(*************************************************************
This function was generated by the 'check array access'
option of the controllers 'properties' dialog box.
If you delete this comment, the 'check array access' option
of the controllers 'properties' dialog box will be removed.
**************************************************************)
    (**************************************************************************************************)
    (* The implementation has to be adjusted to your application/machine.                             *)
    (* This is an exemplary implementation of the function.                                           *)
    (* Per default, an access violation is generated to avoid machine damage                          *)
    (* Check the Call Stack (menu Debug/Callstack) and modify the faulty logic!                       *)
    (**************************************************************************************************)

IF  index < lower THEN 
	errstr:= 'CheckBounds: Lower arrayindex ';
	errstr:=CONCAT(STR1:=errstr  , STR2:= DINT_TO_STRING(lower));
	errstr:=CONCAT(STR1:=errstr  , STR2:= ' underrunned by ');
	errstr:=CONCAT(STR1:=errstr  , STR2:= DINT_TO_STRING(index));
//  This pragma may be removed: 
	{info 'CheckBounds: Please implement your own error reaction below'}
//  EXAMPLE 1 (default): 
//  Set a F0-Error into the diagnostic- and error memory
//  Triggering an access violation --> Application will be stopped and leads to a F5-Error

  ML_SetDiagEntry(
	Severity:= E_LOG_SEVERITY.ERROR, 
	Class:= E_LOG_CLASS.CLASS_0, 
	Facility:= E_LOG_FACILITY.USER, 
	Code:= 0, 
	Text:= ADR(errstr));

	bByte:=ptNull^;(*triggering an access violation *)

// EXAMPLE 2:
// Limit the faulty index to the lower index 
//     -> no memory will be overwritten
//     -> Keep PLC-task and motion running
// Set a E0-Warning into the diagnostic- and error memory
// NOTE: There is still an implementation error in your application code!

//  ML_SetDiagEntry(
//	Severity:= E_LOG_SEVERITY.WARNING, 
//	Class:= E_LOG_CLASS.CLASS_0, 
//	Facility:= E_LOG_FACILITY.USER, 
//	Code:= 0, 
//	Text:= ADR(errstr));
// 
//	CheckBounds := lower; //access to the lower index only 
//  return;
	
ELSIF  index > upper THEN
	errstr:= 'CheckBounds: Higher arrayindex ';
	errstr:=CONCAT(STR1:=errstr  , STR2:= DINT_TO_STRING(upper));
	errstr:=CONCAT(STR1:=errstr  , STR2:= ' overrunned by ');
	errstr:=CONCAT(STR1:=errstr  , STR2:= DINT_TO_STRING(index));

//  this pragma may be removed: 
	{info 'CheckBounds: Please implement your own error reaction below'}
//  example 1 (default): 
//  set a F0-Error into the diagnostic- and error memory
//  triggering an access violation --> Application will be stopped and leads to a F5-Error

  ML_SetDiagEntry(
	Severity:= E_LOG_SEVERITY.ERROR, 
	Class:= E_LOG_CLASS.CLASS_0, 
	Facility:= E_LOG_FACILITY.USER, 
	Code:= 0, 
	Text:= ADR(errstr));

	bByte:=ptNull^;(*triggering an access violation *)

//example 2:
// Limit the faulty index to the upper index 
//     -> no memory will be overwritten
//     -> Keep PLC-task and motion running
// Set a E0-Warning into the diagnostic- and error memory
// NOTE: There is still an implementation error in your application code!

//  ML_SetDiagEntry(
//	Severity:= E_LOG_SEVERITY.WARNING, 
//	Class:= E_LOG_CLASS.CLASS_0, 
//	Facility:= E_LOG_FACILITY.USER, 
//	Code:= 0, 
//	Text:= ADR(errstr));
// 
//	CheckBounds := upper; //access to the upper index only 
//  return;

ELSE // access to array is ok  
	CheckBounds := index;
END_IF

END_FUNCTION

// IndraMotionMlc1/Application/Discrete_FIlter
FUNCTION_BLOCK Discrete_FIlter
VAR_INPUT
	ssMethodType: SINT;
	In: LREAL;
END_VAR
VAR_OUTPUT
	Out: LREAL;
END_VAR
VAR
	DiscreteFilter_states: LREAL;
END_VAR



CASE ssMethodType OF
    0: 
        (* InitializeConditions for DiscreteFilter: '<S1>/Discrete Filter' *)
        DiscreteFilter_states := 0.0;
    1: 
        (* DiscreteFilter: '<S1>/Discrete Filter' *)
        Out := In - (0.5 * DiscreteFilter_states);
        (* Update for DiscreteFilter: '<S1>/Discrete Filter' *)
        DiscreteFilter_states := Out;
END_CASE;

END_FUNCTION_BLOCK

// IndraMotionMlc1/Application/VCC_Anti_DB
PROGRAM VCC_Anti_DB
VAR_INPUT
	u_ref: LREAL;
END_VAR
VAR_OUTPUT
	u_cmd:  LREAL := 6;
END_VAR
VAR
	cyl_extract: LREAL;
	cyl_retract: LREAL;
END_VAR

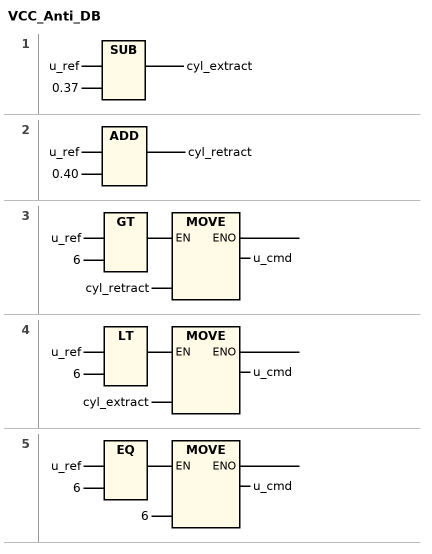
// NETWORK 1
cyl_extract := u_ref - 0.37;

// NETWORK 2
cyl_retract := u_ref + 0.40;

// NETWORK 3
IF u_ref > 6 THEN u_cmd := cyl_retract; END_IF

// NETWORK 4
IF u_ref < 6 THEN u_cmd := cyl_extract; END_IF

// NETWORK 5
IF u_ref = 6 THEN u_cmd := 6; END_IF

END_PROGRAM

// IndraMotionMlc1/Application/S_shape_Profile_old
FUNCTION_BLOCK S_shape_Profile_old
VAR_INPUT
	Enable: BOOL;
	x0: LREAL;
	v0: LREAL;
	Position_SP: LREAL;
	Velocity_SP: LREAL;
	t0: LREAL;
	t_Hold_Position: LREAL;
	CyclicTime: LREAL;
END_VAR
VAR_OUTPUT
	Position_Ref: LREAL;
	Velocity_Ref: LREAL;
	Motion_Cycle_Time: LREAL;
	Error: LREAL;
END_VAR
VAR
	Error_0: DINT;
	jm: LREAL;
	s_acc: LREAL;
	t1: LREAL;
	t2: LREAL;
	t3: LREAL;
	t4: LREAL;
	t5: LREAL;
	t6: LREAL;
	t7: LREAL;
	t8: LREAL;
	t9: LREAL;
	t10: LREAL;
	sh: LREAL;
	vh: LREAL;
	s3: LREAL;
	s4: LREAL;
	v4: LREAL;
	s7: LREAL;
	rtb_Saturation: LREAL;
	rtb_Saturation_tmp: LREAL;
END_VAR


(* Saturate: '<S1>/Saturation' *)

IF Position_SP >= 500.0 THEN 
    rtb_Saturation := 500.0;
ELSIF Position_SP > 0.0 THEN 
    rtb_Saturation := Position_SP;
ELSE 
    rtb_Saturation := 0.0;
END_IF;

(* End of Saturate: '<S1>/Saturation' *)


(* Saturate: '<S1>/Saturation1' *)

IF Velocity_SP >= 150.0 THEN 
    Position_Ref := 150.0;
ELSIF Velocity_SP > -150.0 THEN 
    Position_Ref := Velocity_SP;
ELSE 
    Position_Ref := -150.0;
END_IF;

(* End of Saturate: '<S1>/Saturation1' *)


(* MATLAB Function: '<S1>/SP_Generator' *)
(* MATLAB Function 'S_shape_Profile/SP_Generator': '<S2>:1' *)
(* '<S2>:1:4' PositionSP = Desired_Position - s0; *)
(* '<S2>:1:6' a0 = 0; *)
(* '<S2>:1:7' j0 = 0; *)
(* '<S2>:1:8' AccelerationSP = VelocitySP; *)
(* '<S2>:1:10' vel=VelocitySP; *)
(* '<S2>:1:11' as=AccelerationSP; *)
(* Input velocity  *)
(* '<S2>:1:13' vs=vel; *)
(* [rad/s] *)
(* Delta velocity  *)
(* '<S2>:1:15' dv=(vs-v0); *)
(* [rad/s]      *)
(* Max Jerk Considerations *)
(* '<S2>:1:17' jm=as^2/dv; *)
sh := Position_Ref * Position_Ref;
vh := Position_Ref - v0;
jm := sh / vh;
(* [rad/s^3]  *)
(* Constant Velocity periodes *)
(* '<S2>:1:19' s_acc=(vs^2-v0^2)/as; *)
s_acc := (sh - (v0 * v0)) / Position_Ref;
(* '<S2>:1:20' CstVelTime=(PositionSP-2*s_acc)/vs; *)
rtb_Saturation := ((rtb_Saturation - x0) - (2.0 * s_acc)) / Position_Ref;
(* '<S2>:1:21' if CstVelTime < 0 *)

IF rtb_Saturation < 0.0 THEN 
    (* '<S2>:1:22' Error = 1; *)
    Error_0 := 1;
ELSE 
    (* '<S2>:1:23' else *)
    (* '<S2>:1:24' Error = 0; *)
    Error_0 := 0;
END_IF;

(* Time periodes, *)
(* '<S2>:1:28' t1=t0+(as/jm); *)
s3 := Position_Ref / jm;
t1 := s3 + t0;
(* '<S2>:1:29' t2=t1+(as/jm); *)
t2 := s3 + t1;
(* '<S2>:1:30' t3=t2+CstVelTime; *)
t3 := t2 + rtb_Saturation;
(* '<S2>:1:31' t4=t3+(as/jm); *)
t4 := s3 + t3;
(* '<S2>:1:32' t5=t4+(as/jm); *)
t5 := s3 + t4;
(* '<S2>:1:33' t6=t5+HoldPositionTime; *)
t6 := t5 + t_Hold_Position;
(* '<S2>:1:34' t7=t6+(as/jm); *)
t7 := s3 + t6;
(* '<S2>:1:35' t8=t7+(as/jm); *)
t8 := s3 + t7;
(* '<S2>:1:36' t9=t8+CstVelTime; *)
t9 := t8 + rtb_Saturation;
(* '<S2>:1:37' t10=t9+(as/jm); *)
t10 := s3 + t9;
(* '<S2>:1:38' t11=t10+(as/jm); *)
Motion_Cycle_Time := s3 + t10;
(* Position and Velocity Constants *)
(* '<S2>:1:40' sh=(v0+(as^2)/(6*jm))*(as/jm); *)
sh := ((sh / (6.0 * jm)) + v0) * s3;
(* '<S2>:1:41' vh=(vs-v0)/2; *)
vh := vh / 2.0;
(* '<S2>:1:42' s3=s_acc+vs*(t3-t2); *)
s3 := ((t3 - t2) * Position_Ref) + s_acc;
(* '<S2>:1:43' s4=s3+vs*(t4-t3)-jm*((t4-t3)^3)/6; *)
rtb_Saturation := t4 - t3;
s4 := ((rtb_Saturation * Position_Ref) + s3) - ((EXPT(rtb_Saturation, 3.0) * jm) / 6.0);
(* '<S2>:1:44' v4=vs-jm*((t4-t3)^2)/2; *)
v4 := Position_Ref - (((rtb_Saturation * rtb_Saturation) * jm) / 2.0);
(* '<S2>:1:45' s5=s0+jm*((t5-t4)^3)/6-as*((t5-t4)^2)/2+v4*(t5-t4)+s4; *)
rtb_Saturation_tmp := t5 - t4;
rtb_Saturation := (((((EXPT(rtb_Saturation_tmp, 3.0) * jm) / 6.0) + x0) - (((rtb_Saturation_tmp * rtb_Saturation_tmp) * Position_Ref) / 2.0)) + (rtb_Saturation_tmp * v4)) + s4;
(* s6=s5+(s0+v0*(t7-t6)+jm*((t7-t6)^3)/6); *)
(* '<S2>:1:47' s7= s5-(s_acc+vs*(t9-t8)); *)
s7 := rtb_Saturation - (((t9 - t8) * Position_Ref) + s_acc);
(* '<S2>:1:48' s8= s7-(vs*(t10-t9)-jm*((t10-t9)^3)/6); *)
(* s9= s8-(jm*((t11-t10)^3)/6-as*((t11-t10)^2)/2+v4*(t11-t10)); *)
(* Phase0 *)
(* '<S2>:1:51' if  Error == 1 *)

IF Error_0 = 1 THEN 
    (* '<S2>:1:52' s = s0; *)
    rtb_Saturation := x0;
    (* '<S2>:1:53' v = v0; *)
    Position_Ref := v0;
    (* '<S2>:1:54' a = a0; *)
    (* '<S2>:1:55' j=j0; *)
ELSIF (CyclicTime >= 0.0) AND (CyclicTime <= t0) THEN 
    (* '<S2>:1:56' elseif  (t >= 0) &amp;&amp; (t <= t0) *)
    (* '<S2>:1:57' s = s0; *)
    rtb_Saturation := x0;
    (* '<S2>:1:58' v = v0; *)
    Position_Ref := v0;
    (* '<S2>:1:59' a = a0; *)
    (* '<S2>:1:60' j=j0; *)
    (* Phase1 - concave Acc *)
ELSIF (CyclicTime >= t0) AND (CyclicTime <= t1) THEN 
    (* '<S2>:1:62' elseif  (t >= t0) &amp;&amp; (t <= (t1)) *)
    (* '<S2>:1:63' s = s0+v0*(t-t0)+jm*((t-t0)^3)/6; *)
    rtb_Saturation_tmp := CyclicTime - t0;
    rtb_Saturation := ((rtb_Saturation_tmp * v0) + x0) + ((EXPT(rtb_Saturation_tmp, 3.0) * jm) / 6.0);
    (* '<S2>:1:64' v = v0+jm*((t-t0)^2)/2; *)
    Position_Ref := (((rtb_Saturation_tmp * rtb_Saturation_tmp) * jm) / 2.0) + v0;
    (* '<S2>:1:65' a = jm*(t-t0); *)
    (* '<S2>:1:66' j=jm; *)
    (* Phase2 - convex Acc *)
ELSIF (CyclicTime >= t1) AND (CyclicTime <= t2) THEN 
    (* '<S2>:1:68' elseif (t >= (t1)) &amp;&amp; (t <= (t2)) *)
    (* '<S2>:1:69' s = s0+sh+vh*(t-t1)+as*((t-t1)^2)/2-jm*((t-t1)^3)/6; *)
    rtb_Saturation_tmp := CyclicTime - t1;
    rtb_Saturation := (((rtb_Saturation_tmp * vh) + (x0 + sh)) + (((rtb_Saturation_tmp * rtb_Saturation_tmp) * Position_Ref) / 2.0)) - ((EXPT(rtb_Saturation_tmp, 3.0) * jm) / 6.0);
    (* '<S2>:1:70' v = vh+as*(t-t1)-jm*((t-t1)^2)/2; *)
    Position_Ref := ((rtb_Saturation_tmp * Position_Ref) + vh) - (((rtb_Saturation_tmp * rtb_Saturation_tmp) * jm) / 2.0);
    (* '<S2>:1:71' a = as-jm*(t-t1); *)
    (* '<S2>:1:72' j = -jm; *)
    (* Phase3 - constant velocity *)
ELSIF (CyclicTime >= t2) AND (CyclicTime <= t3) THEN 
    (* '<S2>:1:74' elseif (t >= t2) &amp;&amp; (t <= t3) *)
    (* '<S2>:1:75' s = s0+s_acc+vs*(t-t2); *)
    rtb_Saturation := ((CyclicTime - t2) * Position_Ref) + (x0 + s_acc);
    (* '<S2>:1:76' v = vs; *)
    (* '<S2>:1:77' a = 0; *)
    (* '<S2>:1:78' j = 0; *)
    (* Phase4 - convex Dec *)
ELSIF (CyclicTime >= t3) AND (CyclicTime <= t4) THEN 
    (* '<S2>:1:80' elseif (t >= t3) &amp;&amp; (t <= t4) *)
    (* '<S2>:1:81' s = s0+s3+vs*(t-t3)-jm*((t-t3)^3)/6; *)
    rtb_Saturation_tmp := CyclicTime - t3;
    rtb_Saturation := ((rtb_Saturation_tmp * Position_Ref) + (x0 + s3)) - ((EXPT(rtb_Saturation_tmp, 3.0) * jm) / 6.0);
    (* '<S2>:1:82' v = vs-jm*((t-t3)^2)/2; *)
    Position_Ref := Position_Ref - (((rtb_Saturation_tmp * rtb_Saturation_tmp) * jm) / 2.0);
    (* '<S2>:1:83' a = -jm*(t-t3); *)
    (* '<S2>:1:84' j = -jm; *)
    (* Phase5 - concav Dec *)
ELSIF (CyclicTime >= t4) AND (CyclicTime <= t5) THEN 
    (* '<S2>:1:86' elseif (t >= t4) &amp;&amp; (t <= t5) *)
    (* '<S2>:1:87' s = s0+jm*((t-t4)^3)/6-as*((t-t4)^2)/2+v4*(t-t4)+s4; *)
    rtb_Saturation_tmp := CyclicTime - t4;
    rtb_Saturation := (((((EXPT(rtb_Saturation_tmp, 3.0) * jm) / 6.0) + x0) - (((rtb_Saturation_tmp * rtb_Saturation_tmp) * Position_Ref) / 2.0)) + (rtb_Saturation_tmp * v4)) + s4;
    (* '<S2>:1:88' v = jm*((t-t4)^2)/2-as*(t-t4)+v4; *)
    Position_Ref := ((((rtb_Saturation_tmp * rtb_Saturation_tmp) * jm) / 2.0) - (rtb_Saturation_tmp * Position_Ref)) + v4;
    (* '<S2>:1:89' a = jm*(t-t4)-as; *)
    (* '<S2>:1:90' j=jm; *)
    (* Phase6 - holding position *)
ELSIF (CyclicTime >= t5) AND (CyclicTime <= t6) THEN 
    (* '<S2>:1:92' elseif (t >= t5) &amp;&amp; (t <= t6) *)
    (* '<S2>:1:93' s = s5; *)
    (* '<S2>:1:94' v = 0; *)
    Position_Ref := 0.0;
    (* '<S2>:1:95' a = 0; *)
    (* '<S2>:1:96' j = 0; *)
    (* Phase7 - concave Dec *)
ELSIF (CyclicTime >= t6) AND (CyclicTime <= t7) THEN 
    (* '<S2>:1:98' elseif (t >= t6) &amp;&amp; (t <= t7) *)
    (* '<S2>:1:99' s = s5-(v0*(t-t6)+jm*((t-t6)^3)/6); *)
    rtb_Saturation_tmp := CyclicTime - t6;
    rtb_Saturation := rtb_Saturation - (((EXPT(rtb_Saturation_tmp, 3.0) * jm) / 6.0) + (rtb_Saturation_tmp * v0));
    (* '<S2>:1:100' v = -(v0+jm*((t-t6)^2)/2); *)
    Position_Ref :=  -((((rtb_Saturation_tmp * rtb_Saturation_tmp) * jm) / 2.0) + v0);
    (* '<S2>:1:101' a = -jm*(t-t6); *)
    (* '<S2>:1:102' j=-jm; *)
    (* Phase8 - convex Dec *)
ELSIF (CyclicTime >= t7) AND (CyclicTime <= t8) THEN 
    (* '<S2>:1:104' elseif (t >= t7) &amp;&amp; (t <= t8) *)
    (* '<S2>:1:105' s = s5-(sh+vh*(t-t7)+as*((t-t7)^2)/2-jm*((t-t7)^3)/6); *)
    s3 := CyclicTime - t7;
    rtb_Saturation := rtb_Saturation - ((((s3 * vh) + sh) + (((s3 * s3) * Position_Ref) / 2.0)) - ((EXPT(s3, 3.0) * jm) / 6.0));
    (* '<S2>:1:106' v = -(vh+as*(t-t7)-jm*((t-t7)^2)/2); *)
    Position_Ref :=  -(((s3 * Position_Ref) + vh) - (((s3 * s3) * jm) / 2.0));
    (* '<S2>:1:107' a = -(as-jm*(t-t7)); *)
    (* '<S2>:1:108' j = jm; *)
    (* Phase9 - constant velocity *)
ELSIF (CyclicTime >= t8) AND (CyclicTime <= t9) THEN 
    (* '<S2>:1:110' elseif (t >= t8) &amp;&amp; (t <= t9) *)
    (* '<S2>:1:111' s = s5-(s_acc+vs*(t-t8)); *)
    rtb_Saturation := rtb_Saturation - (((CyclicTime - t8) * Position_Ref) + s_acc);
    (* '<S2>:1:112' v = -vs; *)
    Position_Ref :=  -Position_Ref;
    (* '<S2>:1:113' a = 0; *)
    (* '<S2>:1:114' j = 0; *)
    (* Phase10 - concav Acc *)
ELSIF (CyclicTime >= t9) AND (CyclicTime <= t10) THEN 
    (* '<S2>:1:116' elseif (t >= t9) &amp;&amp; (t <= t10) *)
    (* '<S2>:1:117' s = s7-(vs*(t-t9)-jm*((t-t9)^3)/6); *)
    rtb_Saturation_tmp := CyclicTime - t9;
    rtb_Saturation := s7 - ((rtb_Saturation_tmp * Position_Ref) - ((EXPT(rtb_Saturation_tmp, 3.0) * jm) / 6.0));
    (* '<S2>:1:118' v = -(vs-jm*((t-t9)^2)/2); *)
    Position_Ref :=  -(Position_Ref - (((rtb_Saturation_tmp * rtb_Saturation_tmp) * jm) / 2.0));
    (* '<S2>:1:119' a = jm*(t-t9); *)
    (* '<S2>:1:120' j = jm; *)
    (* Phase11 - convex Acc *)
ELSIF (CyclicTime >= t10) AND (CyclicTime <= Motion_Cycle_Time) THEN 
    (* '<S2>:1:122' elseif (t >= t10) &amp;&amp; (t <= t11) *)
    (* '<S2>:1:123' s = s8-(jm*((t-t10)^3)/6-as*((t-t10)^2)/2+v4*(t-t10)); *)
    rtb_Saturation_tmp := CyclicTime - t10;
    rtb_Saturation := t10 - t9;
    rtb_Saturation := (s7 - ((rtb_Saturation * Position_Ref) - ((EXPT(rtb_Saturation, 3.0) * jm) / 6.0))) - ((((EXPT(rtb_Saturation_tmp, 3.0) * jm) / 6.0) - (((rtb_Saturation_tmp * rtb_Saturation_tmp) * Position_Ref) / 2.0)) + (rtb_Saturation_tmp * v4));
    (* '<S2>:1:124' v = -(jm*((t-t10)^2)/2-as*(t-t10)+v4); *)
    Position_Ref :=  -(((((rtb_Saturation_tmp * rtb_Saturation_tmp) * jm) / 2.0) - (rtb_Saturation_tmp * Position_Ref)) + v4);
    (* '<S2>:1:125' a = -(jm*(t-t10)-as); *)
    (* '<S2>:1:126' j=-jm; *)
    (* Phase12 - hold position *)
ELSE 
    (* '<S2>:1:128' else *)
    (* '<S2>:1:129' s = s0; *)
    rtb_Saturation := x0;
    (* '<S2>:1:130' v = v0; *)
    Position_Ref := v0;
    (* '<S2>:1:131' a = a0; *)
    (* '<S2>:1:132' j = j0; *)
END_IF;

(* '<S2>:1:135' if t == 0 *)

IF CyclicTime = 0.0 THEN 
    (* '<S2>:1:136' PositionRef=s0; *)
    rtb_Saturation := x0;
    (* [mm] *)
END_IF;

(* Switch: '<S1>/Switch' *)
(* '<S2>:1:141' InPositionTime=t11; *)
(* [s] *)
(* '<S2>:1:142' VelocityRef=v; *)
(* [mm/s] *)
(* '<S2>:1:143' AccelerationRef=a; *)
(* [mm/s^2] *)
(* '<S2>:1:144' JerkRef=j; *)
(* %[mm/s^3] *)

IF  NOT Enable THEN 
    Position_Ref := v0;
END_IF;

(* End of Switch: '<S1>/Switch' *)


(* Saturate: '<S1>/Saturation2' *)

IF Position_Ref >= 150.0 THEN 
    (* Outport: '<Root>/Velocity_Ref' *)
    Velocity_Ref := 150.0;
ELSIF Position_Ref > -150.0 THEN 
    (* Outport: '<Root>/Velocity_Ref' *)
    Velocity_Ref := Position_Ref;
ELSE 
    (* Outport: '<Root>/Velocity_Ref' *)
    Velocity_Ref := -150.0;
END_IF;

(* End of Saturate: '<S1>/Saturation2' *)


(* Switch: '<S1>/Switch1' *)

IF Enable THEN 
    Position_Ref := rtb_Saturation;
ELSE 
    Position_Ref := x0;
END_IF;

(* End of Switch: '<S1>/Switch1' *)


(* Saturate: '<S1>/Saturation3' *)

IF Position_Ref >= 500.0 THEN 
    (* Outport: '<Root>/Position_Ref' *)
    Position_Ref := 500.0;
ELSIF  NOT (Position_Ref > 0.0) THEN 
    (* Outport: '<Root>/Position_Ref' *)
    Position_Ref := 0.0;
END_IF;

(* End of Saturate: '<S1>/Saturation3' *)


(* Outport: '<Root>/Error' incorporates:
 *  MATLAB Function: '<S1>/SP_Generator' *)
Error := DINT_TO_LREAL(Error_0);

END_FUNCTION_BLOCK

// IndraMotionMlc1/Application/VCC_Controller_FF_PI_AD_v04
FUNCTION_BLOCK VCC_Controller_FF_PI_AD_v04
VAR_INPUT
	ssMethodType: SINT;
	Tuning_Mode_On: BOOL;
	FB_Cntr_On: BOOL;
	I_Cntr_On: BOOL;
	I_Cntr_Reset_On: BOOL;
	Active_Damper_On: BOOL;
	k_AD_Num: LREAL;
	Pos_Error_Limit: LREAL;
	DB_Up: LREAL;
	DB_Down: LREAL;
	Qmax_Up: LREAL;
	Qmax_Down: LREAL;
	k_P: LREAL;
	k_I: LREAL;
	Pos_Ref: LREAL;
	Vel_Ref: LREAL;
	Pos_FB: LREAL;
	p_A: LREAL;
	p_B: LREAL;
END_VAR
VAR_OUTPUT
	Pos_Error: LREAL;
	u_FF: LREAL;
	u_P: LREAL;
	u_I: LREAL;
	u_AD: LREAL;
	I_reset: LREAL;
	u_DCV: LREAL;
END_VAR
VAR
	rtb_Q_refm3s: LREAL;
	rtb_Saturation1: LREAL;
	rtb_I_Reset: DINT;
	rtb_LoadPressure: LREAL;
	c_DiscreteTimeIntegrator_DS: LREAL;
	VectorConcatenate: ARRAY[0..1] OF LREAL;
	TransferFcn11_states: LREAL;
END_VAR



CASE ssMethodType OF
    0: 
        (* InitializeConditions for DiscreteIntegrator: '<S1>/Discrete-Time Integrator' *)
        c_DiscreteTimeIntegrator_DS := 0.0;
        (* InitializeConditions for DiscreteTransferFcn: '<S4>/Transfer Fcn1 1' *)
        TransferFcn11_states := 0.0;
    1: 
        (* Switch: '<S1>/Switch2' incorporates:
         *  Constant: '<S1>/Annnulus_Area'
         *  Constant: '<S1>/Bore_Area'
         *  Product: '<S1>/Product1'
         *  Product: '<S1>/Product3' *)

        IF Vel_Ref >= 0.0 THEN 
            u_FF := 3318.3 * Vel_Ref;
        ELSE 
            u_FF := Vel_Ref * 2356.2;
        END_IF;

        (* End of Switch: '<S1>/Switch2' *)
        

        (* Gain: '<S1>/Gain2' *)
        rtb_Q_refm3s := 1.0E-9 * u_FF;
        (* Switch: '<S1>/Switch5' *)

        IF Vel_Ref >= 0.0 THEN 
            u_FF := Qmax_Up;
        ELSE 
            u_FF := Qmax_Down;
        END_IF;

        (* End of Switch: '<S1>/Switch5' *)
        

        (* Product: '<S1>/Divide2' incorporates:
         *  Gain: '<S1>/Gain1' *)
        u_FF := (60000.0 * rtb_Q_refm3s) / u_FF;
        (* Sum: '<S1>/Sum1' *)
        Pos_Error := Pos_Ref - Pos_FB;
        (* Product: '<S1>/Product' *)
        u_P := k_P * Pos_Error;
        (* MATLAB Function: '<S1>/Controller_Reset' *)
        (* MATLAB Function 'VCC_Controller_FF_PI_AD_v04/Controller_Reset': '<S3>:1' *)
        (* '<S3>:1:3' I_Reset = 1; *)
        (* '<S3>:1:5' if (abs(Pos_Error) <= Pos_Error_Limit) &amp;&amp; (Vel_SP == 0) *)

        IF ABS(Pos_Error) <= Pos_Error_Limit THEN 

            IF Vel_Ref = 0.0 THEN 
                (* '<S3>:1:6' I_Reset = 1; *)
                rtb_I_Reset := 1;
            ELSE 
                (* '<S3>:1:7' else *)
                (* '<S3>:1:8' I_Reset = 0; *)
                rtb_I_Reset := 0;
            END_IF;

        ELSE 
            (* '<S3>:1:7' else *)
            (* '<S3>:1:8' I_Reset = 0; *)
            rtb_I_Reset := 0;
        END_IF;

        (* End of MATLAB Function: '<S1>/Controller_Reset' *)
        

        (* Switch: '<S1>/Switch3' incorporates:
         *  Constant: '<S1>/Constant2' *)

        IF I_Cntr_Reset_On THEN 
            I_reset := DINT_TO_LREAL(rtb_I_Reset);
        ELSE 
            I_reset := 0.0;
        END_IF;

        (* End of Switch: '<S1>/Switch3' *)
        

        (* DiscreteIntegrator: '<S1>/Discrete-Time Integrator' *)

        IF I_reset <> 0.0 THEN 
            c_DiscreteTimeIntegrator_DS := 0.0;
        END_IF;

        (* SignalConversion: '<S4>/ConcatBufferAtVector ConcatenateIn1' *)
        VectorConcatenate[0] := k_AD_Num;
        (* Gain: '<S4>/Gain1' *)
        VectorConcatenate[1] :=  -k_AD_Num;
        (* DiscreteTransferFcn: '<S4>/Transfer Fcn1 1' incorporates:
         *  Gain: '<S4>/Cylinder Area Ratio'
         *  Sum: '<S4>/Load Pressure' *)
        rtb_Q_refm3s := (p_A - (0.710059171597633 * p_B)) - (-0.997 * TransferFcn11_states);
        u_AD := (VectorConcatenate[0] * rtb_Q_refm3s) + (VectorConcatenate[1] * TransferFcn11_states);
        (* Switch: '<S1>/Switch' incorporates:
         *  Constant: '<S1>/Constant'
         *  DiscreteIntegrator: '<S1>/Discrete-Time Integrator' *)

        IF I_Cntr_On THEN 
            u_I := c_DiscreteTimeIntegrator_DS;
        ELSE 
            u_I := 0.0;
        END_IF;

        (* End of Switch: '<S1>/Switch' *)
        

        (* Switch: '<S1>/Switch1' incorporates:
         *  Constant: '<S1>/Constant1'
         *  Sum: '<S1>/Sum5' *)

        IF FB_Cntr_On THEN 
            rtb_LoadPressure := u_P + u_I;
        ELSE 
            rtb_LoadPressure := 0.0;
        END_IF;

        (* End of Switch: '<S1>/Switch1' *)
        

        (* Saturate: '<S1>/Saturation1' *)

        IF rtb_LoadPressure >= 1.0 THEN 
            rtb_Saturation1 := 1.0;
        ELSIF rtb_LoadPressure > -1.0 THEN 
            rtb_Saturation1 := rtb_LoadPressure;
        ELSE 
            rtb_Saturation1 := -1.0;
        END_IF;

        (* End of Saturate: '<S1>/Saturation1' *)
        

        (* Switch: '<S1>/Switch4' incorporates:
         *  Constant: '<S1>/Constant3' *)

        IF  NOT Active_Damper_On THEN 
            u_AD := 0.0;
        END_IF;

        (* End of Switch: '<S1>/Switch4' *)
        

        (* Gain: '<S1>/Gain' incorporates:
         *  Sum: '<S1>/Sum6' *)
        u_DCV :=  -((u_FF + rtb_Saturation1) - u_AD);
        (* Saturate: '<S1>/Saturation5' *)

        IF u_DCV >= 1.0 THEN 
            u_DCV := 1.0;
        ELSIF  NOT (u_DCV > -1.0) THEN 
            u_DCV := -1.0;
        END_IF;

        (* End of Saturate: '<S1>/Saturation5' *)
        

        (* MATLAB Function: '<S1>/Anti_Dead_Band' *)
        (* MATLAB Function 'VCC_Controller_FF_PI_AD_v04/Anti_Dead_Band': '<S2>:1' *)
        (* '<S2>:1:5' u_DCV = 0; *)
        (* '<S2>:1:7' if (I_Reset == 1) &amp;&amp; (Tuning_Mode == 0) *)

        IF (rtb_I_Reset = 1) AND ( NOT Tuning_Mode_On) THEN 
            (* Outport: '<Root>/u_DCV' *)
            (* '<S2>:1:8' u_DCV = 0; *)
            u_DCV := 0.0;
        ELSIF u_DCV < -0.001 THEN 
            (* Outport: '<Root>/u_DCV' *)
            (* '<S2>:1:9' elseif (u_DCV_ref < -0.001) *)
            (* '<S2>:1:10' u_DCV = -DB_Up + (1-DB_Up)*u_DCV_ref; *)
            u_DCV := ((1.0 - DB_Up) * u_DCV) + ( -DB_Up);
        ELSIF u_DCV > 0.001 THEN 
            (* Outport: '<Root>/u_DCV' *)
            (* '<S2>:1:11' elseif (u_DCV_ref > 0.001) *)
            (* '<S2>:1:12' u_DCV = DB_Down + (1-DB_Down)*u_DCV_ref; *)
            u_DCV := ((1.0 - DB_Down) * u_DCV) + DB_Down;
        ELSE 
            (* Outport: '<Root>/u_DCV' *)
            (* '<S2>:1:13' else *)
            (* '<S2>:1:14' u_DCV = 0; *)
            u_DCV := 0.0;
        END_IF;

        (* End of MATLAB Function: '<S1>/Anti_Dead_Band' *)
        

        (* Update for DiscreteIntegrator: '<S1>/Discrete-Time Integrator' incorporates:
         *  Product: '<S1>/Divide'
         *  Product: '<S1>/Product2'
         *  Sum: '<S1>/Sum2'
         *  Sum: '<S1>/Sum3' *)
        c_DiscreteTimeIntegrator_DS := (((((rtb_Saturation1 - rtb_LoadPressure) / k_P) + Pos_Error) * k_I) * 0.001) + c_DiscreteTimeIntegrator_DS;
        (* Update for DiscreteTransferFcn: '<S4>/Transfer Fcn1 1' *)
        TransferFcn11_states := rtb_Q_refm3s;
END_CASE;

END_FUNCTION_BLOCK

// IndraMotionMlc1/Application/ZCFCN_d_ANY
FUNCTION_BLOCK ZCFCN_d_ANY
VAR_INPUT
	u0: USINT;
	u1: LREAL;
END_VAR
VAR_OUTPUT
	y0: DINT;
	y1: USINT;
END_VAR
VAR
	rising: BOOL;
	temp1: BOOL;
	falling: BOOL;
	temp2: BOOL;
END_VAR


temp1 := FALSE;

IF u1 > 0.0 THEN 
    y1 := 1;
ELSIF u1 < 0.0 THEN 
    y1 := 2;
ELSE 
    y1 := 0;
END_IF;

temp2 := FALSE;

IF u0 = 2 THEN 

    IF y1 = 0 THEN 
        rising := TRUE;
    ELSIF y1 = 1 THEN 
        rising := TRUE;
    ELSE 
        temp2 := TRUE;
    END_IF;

ELSE 
    temp2 := TRUE;
END_IF;


IF temp2 THEN 

    IF u0 = 0 THEN 

        IF y1 = 1 THEN 
            rising := TRUE;
        ELSE 
            temp1 := TRUE;
        END_IF;

    ELSE 
        temp1 := TRUE;
    END_IF;

END_IF;


IF temp1 THEN 

    IF u0 = 101 THEN 

        IF y1 = 1 THEN 
            rising := TRUE;
        ELSE 
            rising := FALSE;
        END_IF;

    ELSE 
        rising := FALSE;
    END_IF;

END_IF;


IF rising THEN 
    y0 := 1;
ELSE 
    temp1 := FALSE;
    temp2 := FALSE;

    IF u0 = 1 THEN 

        IF y1 = 0 THEN 
            falling := TRUE;
        ELSIF y1 = 2 THEN 
            falling := TRUE;
        ELSE 
            temp2 := TRUE;
        END_IF;

    ELSE 
        temp2 := TRUE;
    END_IF;


    IF temp2 THEN 

        IF u0 = 0 THEN 

            IF y1 = 2 THEN 
                falling := TRUE;
            ELSE 
                temp1 := TRUE;
            END_IF;

        ELSE 
            temp1 := TRUE;
        END_IF;

    END_IF;


    IF temp1 THEN 

        IF u0 = 100 THEN 

            IF y1 = 2 THEN 
                falling := TRUE;
            ELSE 
                falling := FALSE;
            END_IF;

        ELSE 
            falling := FALSE;
        END_IF;

    END_IF;


    IF falling THEN 
        y0 := -1;
    ELSE 
        y0 := 0;
    END_IF;

END_IF;


IF (u0 = 2) AND (y1 = 0) THEN 
    y1 := 100;
ELSIF (u0 = 1) AND (y1 = 0) THEN 
    y1 := 101;
END_IF;

END_FUNCTION_BLOCK

// IndraMotionMlc1/Application/Primary_Control2
FUNCTION_BLOCK Primary_Control2
VAR_INPUT
	b_time: LREAL;
	xref2: LREAL;
	x: LREAL;
	pA: LREAL;
	pB: LREAL;
END_VAR
VAR_OUTPUT
	disc_time: LREAL;
	wmref: LREAL;
	wmref_sat: LREAL;
	xref: LREAL;
	dxref: LREAL;
	ddxref: LREAL;
	Pos_error: LREAL;
	dxref_operator: LREAL;
	dxref_lim: LREAL;
END_VAR
VAR
	rate: LREAL;
	e: LREAL;
	uHP: LREAL;
	ui: LREAL;
	ei: LREAL;
	uiold_not_empty: BOOL;
	eiold: LREAL;
	dxref_lim_old: LREAL;
	xref_old: LREAL;
	wmref_sat_old: LREAL;
	ddxref_old: LREAL;
	ddxref_oldold: LREAL;
	dxref_lim_oldold: LREAL;
	dxref_old: LREAL;
	dxref_oldold: LREAL;
	wmref_old: LREAL;
	pLold: LREAL;
	uHPold: LREAL;
	uiold: LREAL;
	wm_ini: LREAL := 0.62103355053102638;
	x_ini: LREAL := 0.05;
	pA_ini: LREAL := 6.9337754512426769E+6;
	A_B: LREAL := 0.0023561944901923449;
	A_A: LREAL := 0.0033183072403542195;
	pB_ini: LREAL := 80830.0;
	Txm22: LREAL := 0.001;
	slew_limit_ref: LREAL := 0.10447093700391079;
	w_input: LREAL := 6.2831853071795862;
	wad: LREAL := 18.849555921538759;
	Cawx: LREAL := 16.666666666666664;
	Cix: LREAL := 3141.5926535897929;
	Cff: LREAL := 2004.7633939712759;
	Cpx: LREAL := 942.47779607693792;
	Cad: LREAL := 5.2359877559829886E-6;
	wm_lim: LREAL := 376.99111843077515;
	need_init: BOOL := TRUE;
END_VAR



IF need_init THEN 
    (* SystemInitialize for MATLAB Function: '<Root>/Primary_Control2' *)
    uiold_not_empty := FALSE;
    uiold := 0.0;
    dxref_lim_old := 0.0;
    dxref_lim_oldold := 0.0;
    dxref_old := 0.0;
    dxref_oldold := 0.0;
    ddxref_old := 0.0;
    ddxref_oldold := 0.0;
    uHPold := 0.0;
    need_init := FALSE;
END_IF;

(* MATLAB Function: '<Root>/Primary_Control2' *)
(* Motion controller (primary control) for SHA-type drive - Lasse Schmidt, ET/AAU - Date: 11-11-2020 *)
(* MATLAB Function 'Primary_Control2': '<S1>:1' *)
(* '<S1>:1:4' disc_time = time; *)
(* Sample time for control device *)
(* '<S1>:1:6' T=Txm22; *)
(* Initialization of variables *)

(* '<S1>:1:10' if isempty(uiold) *)

IF  NOT uiold_not_empty THEN 
    (* '<S1>:1:11' uiold = 0; *)
    uiold_not_empty := TRUE;
    (* '<S1>:1:12' eiold = wm_ini; *)
    eiold := wm_ini;
    (* '<S1>:1:13' dxref_lim_old = 0; *)
    (* '<S1>:1:14' dxref_lim_oldold = 0; *)
    (* '<S1>:1:15' dxref_old = 0; *)
    (* '<S1>:1:16' dxref_oldold = 0; *)
    (* '<S1>:1:17' ddxref_old = 0; *)
    (* '<S1>:1:18' ddxref_oldold = 0; *)
    (* '<S1>:1:19' xref_old = x_ini; *)
    xref_old := x_ini;
    (* '<S1>:1:20' wmref_sat_old = wm_ini; *)
    wmref_sat_old := wm_ini;
    (* '<S1>:1:21' wmref_old = wm_ini; *)
    wmref_old := wm_ini;
    (* '<S1>:1:22' pLold = (pA_ini-A_B/A_A*pB_ini); *)
    pLold := pA_ini - ((A_B / A_A) * pB_ini);
    (* '<S1>:1:23' uHPold = 0; *)
END_IF;

(* Reference generation *)
(* "Operator input" *)
(* '<S1>:1:27' k = 150/80; *)

(* '<S1>:1:28' dxref_operator = (time>=0)*(time<5/k)*0 + (time>=5/k)*(time<2*5/k)*80*k/1000 + (time>=2*5/k)*(time<4*5/k)*0 - (time>=4*5/k)*(time<5*5/k)*80*k/1000; *)
dxref_operator := (((DINT_TO_LREAL(BOOL_TO_DINT(b_time >= 2.6666666666666665) * BOOL_TO_DINT(b_time < 5.333333333333333)) * 80.0) * 1.875) / 1000.0) - (((DINT_TO_LREAL(BOOL_TO_DINT(b_time >= 10.666666666666666) * BOOL_TO_DINT(b_time < 13.333333333333334)) * 80.0) * 1.875) / 1000.0);
(* Rate limiter for of operator input *)
(* '<S1>:1:30' rate = (dxref_operator-dxref_lim_old)/Txm22; *)
rate := (dxref_operator - dxref_lim_old) / Txm22;
(* Limited rate of operator input *)
(* '<S1>:1:32' if abs(rate)<=slew_limit_ref *)

IF ABS(rate) > slew_limit_ref THEN 
    (* '<S1>:1:34' else *)
    (* '<S1>:1:35' F = slew_limit_ref*sign(rate); *)

    IF rate < 0.0 THEN 
        rate := -1.0;
    ELSIF rate > 0.0 THEN 
        rate := 1.0;
    END_IF;

    rate := slew_limit_ref * rate;
END_IF;

(* Limited "Operator input" *)
(* '<S1>:1:38' dxref_lim = F*T+dxref_lim_old; *)
dxref_lim := (rate * Txm22) + dxref_lim_old;
(* Limited and filtered reference(s) *)
(* '<S1>:1:40' ddxref = -(2*T^2*w_input^2*ddxref_old+T^2*w_input^2*ddxref_oldold-2*T*w_input^2*dxref_lim+2*T*w_input^2*dxref_lim_oldold-4*T*w_input*ddxref_oldold-8*ddxref_old+4*ddxref_oldold)/(T*w_input+2)^2; *)
rate := (Txm22 * w_input) + 2.0;
uHP := Txm22 * Txm22;
ui := w_input * w_input;
e := (2.0 * Txm22) * ui;
ei := (uHP * 2.0) * ui;
uHP := uHP * ui;
ui := (4.0 * Txm22) * w_input;
ddxref := ( -(((((((ei * ddxref_old) + (uHP * ddxref_oldold)) - (e * dxref_lim)) + (e * dxref_lim_oldold)) - (ui * ddxref_oldold)) - (8.0 * ddxref_old)) + (4.0 * ddxref_oldold))) / (rate * rate);
(* '<S1>:1:41' dxref = (T^2*w_input^2*dxref_lim+2*T^2*w_input^2*dxref_lim_old-2*T^2*w_input^2*dxref_old-T^2*w_input^2*dxref_oldold+T^2*w_input^2*dxref_lim_oldold+4*T*w_input*dxref_oldold+8*dxref_old-4*dxref_oldold)/(T*w_input+2)^2; *)
dxref := ((((((((ei * dxref_lim_old) + (uHP * dxref_lim)) - (ei * dxref_old)) - (uHP * dxref_oldold)) + (uHP * dxref_lim_oldold)) + (ui * dxref_oldold)) + (8.0 * dxref_old)) - (4.0 * dxref_oldold)) / (rate * rate);
(* '<S1>:1:42' xref = T/2*(dxref+dxref_old)+xref_old; *)
xref := ((Txm22 / 2.0) * (dxref + dxref_old)) + xref_old;
(* Controller - discrete implementation by forward euler transform *)
(* States used in motion controller *)
(* '<S1>:1:45' pL = pA - A_B/A_A*pB; *)
rate := pA - ((A_B / A_A) * pB);
(* '<S1>:1:46' e = xref2-x; *)
e := xref2 - x;
(* Output of high-pass pressure filter *)
(* '<S1>:1:48' if time > 0 *)

IF b_time > 0.0 THEN 
    (* '<S1>:1:49' uHP = -(T*wad*uHPold-2*pL+2*pLold-2*uHPold)/(T*wad+2); *)
    uHP := Txm22 * wad;
    uHP := ( -((((uHP * uHPold) - (2.0 * rate)) + (2.0 * pLold)) - (2.0 * uHPold))) / (uHP + 2.0);
    (* Input to integral control term *)
    (* '<S1>:1:57' ui = (e - Cawx*(wmref_old-wmref_sat_old))*Cix; *)
    ui := (e - ((wmref_old - wmref_sat_old) * Cawx)) * Cix;
    (* Output of integral term of PI controller with anti wind-up loop *)
    (* '<S1>:1:59' ei = T/2*(ui+uiold)+eiold; *)
    ei := ((Txm22 / 2.0) * (ui + uiold)) + eiold;
ELSE 
    (* '<S1>:1:50' else *)
    (* '<S1>:1:51' uHP = 0; *)
    uHP := 0.0;
    (* '<S1>:1:60' else *)
    (* '<S1>:1:61' ui = 0; *)
    ui := 0.0;
    (* '<S1>:1:62' ei = 0; *)
    ei := 0.0;
END_IF;

(* Integral control part  *)
(* '<S1>:1:55' if time > 0 *)
(* E-motor speed reference *)
(* '<S1>:1:65' wmref = Cff*dxref + Cpx*e + ei - Cad*uHP; *)
wmref := (((Cff * dxref) + (Cpx * e)) + ei) - (Cad * uHP);
(* Limited E-motor speed reference *)
(* '<S1>:1:67' if abs(wmref)<=wm_lim *)

IF ABS(wmref) <= wm_lim THEN 
    (* '<S1>:1:68' wmref_sat = wmref; *)
    wmref_sat := wmref;
ELSE 
    (* '<S1>:1:69' else *)
    (* '<S1>:1:70' wmref_sat = wm_lim*sign(wmref); *)

    IF wmref < 0.0 THEN 
        e := -1.0;
    ELSIF wmref > 0.0 THEN 
        e := 1.0;
    ELSE 
        e := wmref;
    END_IF;

    wmref_sat := wm_lim * e;
END_IF;

(* Delayed states *)
(* '<S1>:1:73' uHPold=uHP; *)
uHPold := uHP;
(* '<S1>:1:74' pLold=pL; *)
pLold := rate;
(* '<S1>:1:75' eiold=ei; *)
eiold := ei;
(* '<S1>:1:76' uiold=ui; *)
uiold := ui;
(* '<S1>:1:77' dxref_lim_oldold=dxref_lim_old; *)
dxref_lim_oldold := dxref_lim_old;
(* '<S1>:1:78' dxref_lim_old=dxref_lim; *)
dxref_lim_old := dxref_lim;
(* '<S1>:1:79' dxref_oldold=dxref_old; *)
dxref_oldold := dxref_old;
(* '<S1>:1:80' dxref_old=dxref; *)
dxref_old := dxref;
(* '<S1>:1:81' ddxref_oldold = ddxref_old; *)
ddxref_oldold := ddxref_old;
(* '<S1>:1:82' ddxref_old = ddxref; *)
ddxref_old := ddxref;
(* '<S1>:1:83' xref_old = xref; *)
xref_old := xref;
(* '<S1>:1:84' wmref_sat_old = wmref_sat; *)
wmref_sat_old := wmref_sat;
(* '<S1>:1:85' wmref_old = wmref; *)
wmref_old := wmref;
(* Outport: '<Root>/disc_time' incorporates:
 *  MATLAB Function: '<Root>/Primary_Control2' *)
(* Position error *)
(* '<S1>:1:87' Pos_error = xref-x; *)
(* End *)
disc_time := b_time;
(* Outport: '<Root>/Pos_error' incorporates:
 *  MATLAB Function: '<Root>/Primary_Control2' *)
Pos_error := xref - x;

END_FUNCTION_BLOCK

// IndraMotionMlc1/Application/Primary_Control1
FUNCTION_BLOCK Primary_Control1
VAR_INPUT
	b_time: LREAL;
	x: LREAL;
	pA: LREAL;
	pB: LREAL;
END_VAR
VAR_OUTPUT
	disc_time: LREAL;
	wmref: LREAL;
	wmref_sat: LREAL;
	xref: LREAL;
	dxref: LREAL;
	ddxref: LREAL;
	Pos_error: LREAL;
	dxref_operator: LREAL;
	dxref_lim: LREAL;
END_VAR
VAR
	rate: LREAL;
	uHP: LREAL;
	ui: LREAL;
	ei: LREAL;
	ddxref_tmp: LREAL;
	uiold_not_empty: BOOL;
	eiold: LREAL;
	dxref_lim_old: LREAL;
	xref_old: LREAL;
	wmref_sat_old: LREAL;
	ddxref_old: LREAL;
	ddxref_oldold: LREAL;
	dxref_lim_oldold: LREAL;
	dxref_old: LREAL;
	dxref_oldold: LREAL;
	wmref_old: LREAL;
	pLold: LREAL;
	uHPold: LREAL;
	uiold: LREAL;
	wm_ini: LREAL := 0.62103355053102638;
	x_ini: LREAL := 0.05;
	pA_ini: LREAL := 6.9337754512426769E+6;
	A_B: LREAL := 0.0023561944901923449;
	A_A: LREAL := 0.0033183072403542195;
	pB_ini: LREAL := 80830.0;
	Txm22: LREAL := 0.001;
	slew_limit_ref: LREAL := 0.10447093700391079;
	w_input: LREAL := 6.2831853071795862;
	wad: LREAL := 18.849555921538759;
	Cawx: LREAL := 16.666666666666664;
	Cix: LREAL := 3141.5926535897929;
	Cff: LREAL := 2004.7633939712759;
	Cpx: LREAL := 942.47779607693792;
	Cad: LREAL := 5.2359877559829886E-6;
	wm_lim: LREAL := 376.99111843077515;
	need_init: BOOL := TRUE;
END_VAR



IF need_init THEN 
    (* SystemInitialize for MATLAB Function: '<Root>/Primary_Control1' *)
    uiold_not_empty := FALSE;
    uiold := 0.0;
    dxref_lim_old := 0.0;
    dxref_lim_oldold := 0.0;
    dxref_old := 0.0;
    dxref_oldold := 0.0;
    ddxref_old := 0.0;
    ddxref_oldold := 0.0;
    uHPold := 0.0;
    need_init := FALSE;
END_IF;

(* MATLAB Function: '<Root>/Primary_Control1' *)
(* Motion controller (primary control) for SHA-type drive - Lasse Schmidt, ET/AAU - Date: 11-11-2020 *)
(* MATLAB Function 'Primary_Control1': '<S1>:1' *)
(* '<S1>:1:4' disc_time = time; *)
(* Sample time for control device *)
(* '<S1>:1:6' T=Txm22; *)
(* Initialization of variables *)

(* '<S1>:1:10' if isempty(uiold) *)

IF  NOT uiold_not_empty THEN 
    (* '<S1>:1:11' uiold = 0; *)
    uiold_not_empty := TRUE;
    (* '<S1>:1:12' eiold = wm_ini; *)
    eiold := wm_ini;
    (* '<S1>:1:13' dxref_lim_old = 0; *)
    (* '<S1>:1:14' dxref_lim_oldold = 0; *)
    (* '<S1>:1:15' dxref_old = 0; *)
    (* '<S1>:1:16' dxref_oldold = 0; *)
    (* '<S1>:1:17' ddxref_old = 0; *)
    (* '<S1>:1:18' ddxref_oldold = 0; *)
    (* '<S1>:1:19' xref_old = x_ini; *)
    xref_old := x_ini;
    (* '<S1>:1:20' wmref_sat_old = wm_ini; *)
    wmref_sat_old := wm_ini;
    (* '<S1>:1:21' wmref_old = wm_ini; *)
    wmref_old := wm_ini;
    (* '<S1>:1:22' pLold = (pA_ini-A_B/A_A*pB_ini); *)
    pLold := pA_ini - ((A_B / A_A) * pB_ini);
    (* '<S1>:1:23' uHPold = 0; *)
END_IF;

(* Reference generation *)
(* "Operator input" *)
(* '<S1>:1:27' k = 150/80; *)

(* '<S1>:1:28' dxref_operator = (time>=0)*(time<5/k)*0 + (time>=5/k)*(time<2*5/k)*80*k/1000 + (time>=2*5/k)*(time<4*5/k)*0 - (time>=4*5/k)*(time<5*5/k)*80*k/1000; *)
dxref_operator := (((DINT_TO_LREAL(BOOL_TO_DINT(b_time >= 2.6666666666666665) * BOOL_TO_DINT(b_time < 5.333333333333333)) * 80.0) * 1.875) / 1000.0) - (((DINT_TO_LREAL(BOOL_TO_DINT(b_time >= 10.666666666666666) * BOOL_TO_DINT(b_time < 13.333333333333334)) * 80.0) * 1.875) / 1000.0);
(* Rate limiter for of operator input *)
(* '<S1>:1:30' rate = (dxref_operator-dxref_lim_old)/Txm22; *)
rate := (dxref_operator - dxref_lim_old) / Txm22;
(* Limited rate of operator input *)
(* '<S1>:1:32' if abs(rate)<=slew_limit_ref *)

IF ABS(rate) > slew_limit_ref THEN 
    (* '<S1>:1:34' else *)
    (* '<S1>:1:35' F = slew_limit_ref*sign(rate); *)

    IF rate < 0.0 THEN 
        rate := -1.0;
    ELSIF rate > 0.0 THEN 
        rate := 1.0;
    END_IF;

    rate := slew_limit_ref * rate;
END_IF;

(* Limited "Operator input" *)
(* '<S1>:1:38' dxref_lim = F*T+dxref_lim_old; *)
dxref_lim := (rate * Txm22) + dxref_lim_old;
(* Limited and filtered reference(s) *)
(* '<S1>:1:40' ddxref = -(2*T^2*w_input^2*ddxref_old+T^2*w_input^2*ddxref_oldold-2*T*w_input^2*dxref_lim+2*T*w_input^2*dxref_lim_oldold-4*T*w_input*ddxref_oldold-8*ddxref_old+4*ddxref_oldold)/(T*w_input+2)^2; *)
rate := (Txm22 * w_input) + 2.0;
uHP := Txm22 * Txm22;
ui := w_input * w_input;
ddxref_tmp := (2.0 * Txm22) * ui;
ei := (uHP * 2.0) * ui;
uHP := uHP * ui;
ui := (4.0 * Txm22) * w_input;
ddxref := ( -(((((((ei * ddxref_old) + (uHP * ddxref_oldold)) - (ddxref_tmp * dxref_lim)) + (ddxref_tmp * dxref_lim_oldold)) - (ui * ddxref_oldold)) - (8.0 * ddxref_old)) + (4.0 * ddxref_oldold))) / (rate * rate);
(* '<S1>:1:41' dxref = (T^2*w_input^2*dxref_lim+2*T^2*w_input^2*dxref_lim_old-2*T^2*w_input^2*dxref_old-T^2*w_input^2*dxref_oldold+T^2*w_input^2*dxref_lim_oldold+4*T*w_input*dxref_oldold+8*dxref_old-4*dxref_oldold)/(T*w_input+2)^2; *)
dxref := ((((((((ei * dxref_lim_old) + (uHP * dxref_lim)) - (ei * dxref_old)) - (uHP * dxref_oldold)) + (uHP * dxref_lim_oldold)) + (ui * dxref_oldold)) + (8.0 * dxref_old)) - (4.0 * dxref_oldold)) / (rate * rate);
(* '<S1>:1:42' xref = T/2*(dxref+dxref_old)+xref_old; *)
xref := ((Txm22 / 2.0) * (dxref + dxref_old)) + xref_old;
(* Controller - discrete implementation by forward euler transform *)
(* States used in motion controller *)
(* '<S1>:1:45' pL = pA - A_B/A_A*pB; *)
rate := pA - ((A_B / A_A) * pB);
(* '<S1>:1:46' e = xref-x; *)
Pos_error := xref - x;
(* Output of high-pass pressure filter *)
(* '<S1>:1:48' if time > 0 *)

IF b_time > 0.0 THEN 
    (* '<S1>:1:49' uHP = -(T*wad*uHPold-2*pL+2*pLold-2*uHPold)/(T*wad+2); *)
    uHP := Txm22 * wad;
    uHP := ( -((((uHP * uHPold) - (2.0 * rate)) + (2.0 * pLold)) - (2.0 * uHPold))) / (uHP + 2.0);
    (* Input to integral control term *)
    (* '<S1>:1:57' ui = (e - Cawx*(wmref_old-wmref_sat_old))*Cix; *)
    ui := (Pos_error - ((wmref_old - wmref_sat_old) * Cawx)) * Cix;
    (* Output of integral term of PI controller with anti wind-up loop *)
    (* '<S1>:1:59' ei = T/2*(ui+uiold)+eiold; *)
    ei := ((Txm22 / 2.0) * (ui + uiold)) + eiold;
ELSE 
    (* '<S1>:1:50' else *)
    (* '<S1>:1:51' uHP = 0; *)
    uHP := 0.0;
    (* '<S1>:1:60' else *)
    (* '<S1>:1:61' ui = 0; *)
    ui := 0.0;
    (* '<S1>:1:62' ei = 0; *)
    ei := 0.0;
END_IF;

(* Integral control part  *)
(* '<S1>:1:55' if time > 0 *)
(* E-motor speed reference *)
(* '<S1>:1:65' wmref = Cff*dxref + Cpx*e + ei - Cad*uHP; *)
wmref := (((Cff * dxref) + (Cpx * Pos_error)) + ei) - (Cad * uHP);
(* Limited E-motor speed reference *)
(* '<S1>:1:67' if abs(wmref)<=wm_lim *)

IF ABS(wmref) <= wm_lim THEN 
    (* '<S1>:1:68' wmref_sat = wmref; *)
    wmref_sat := wmref;
ELSE 
    (* '<S1>:1:69' else *)
    (* '<S1>:1:70' wmref_sat = wm_lim*sign(wmref); *)

    IF wmref < 0.0 THEN 
        ddxref_tmp := -1.0;
    ELSIF wmref > 0.0 THEN 
        ddxref_tmp := 1.0;
    ELSE 
        ddxref_tmp := wmref;
    END_IF;

    wmref_sat := wm_lim * ddxref_tmp;
END_IF;

(* Delayed states *)
(* '<S1>:1:73' uHPold=uHP; *)
uHPold := uHP;
(* '<S1>:1:74' pLold=pL; *)
pLold := rate;
(* '<S1>:1:75' eiold=ei; *)
eiold := ei;
(* '<S1>:1:76' uiold=ui; *)
uiold := ui;
(* '<S1>:1:77' dxref_lim_oldold=dxref_lim_old; *)
dxref_lim_oldold := dxref_lim_old;
(* '<S1>:1:78' dxref_lim_old=dxref_lim; *)
dxref_lim_old := dxref_lim;
(* '<S1>:1:79' dxref_oldold=dxref_old; *)
dxref_oldold := dxref_old;
(* '<S1>:1:80' dxref_old=dxref; *)
dxref_old := dxref;
(* '<S1>:1:81' ddxref_oldold = ddxref_old; *)
ddxref_oldold := ddxref_old;
(* '<S1>:1:82' ddxref_old = ddxref; *)
ddxref_old := ddxref;
(* '<S1>:1:83' xref_old = xref; *)
xref_old := xref;
(* '<S1>:1:84' wmref_sat_old = wmref_sat; *)
wmref_sat_old := wmref_sat;
(* '<S1>:1:85' wmref_old = wmref; *)
wmref_old := wmref;
(* Outport: '<Root>/disc_time' incorporates:
 *  MATLAB Function: '<Root>/Primary_Control1' *)
(* Position error *)
(* '<S1>:1:87' Pos_error = xref-x; *)
(* End *)
disc_time := b_time;

END_FUNCTION_BLOCK

// IndraMotionMlc1/Application/Visualization/VCC/VCC_Visualization
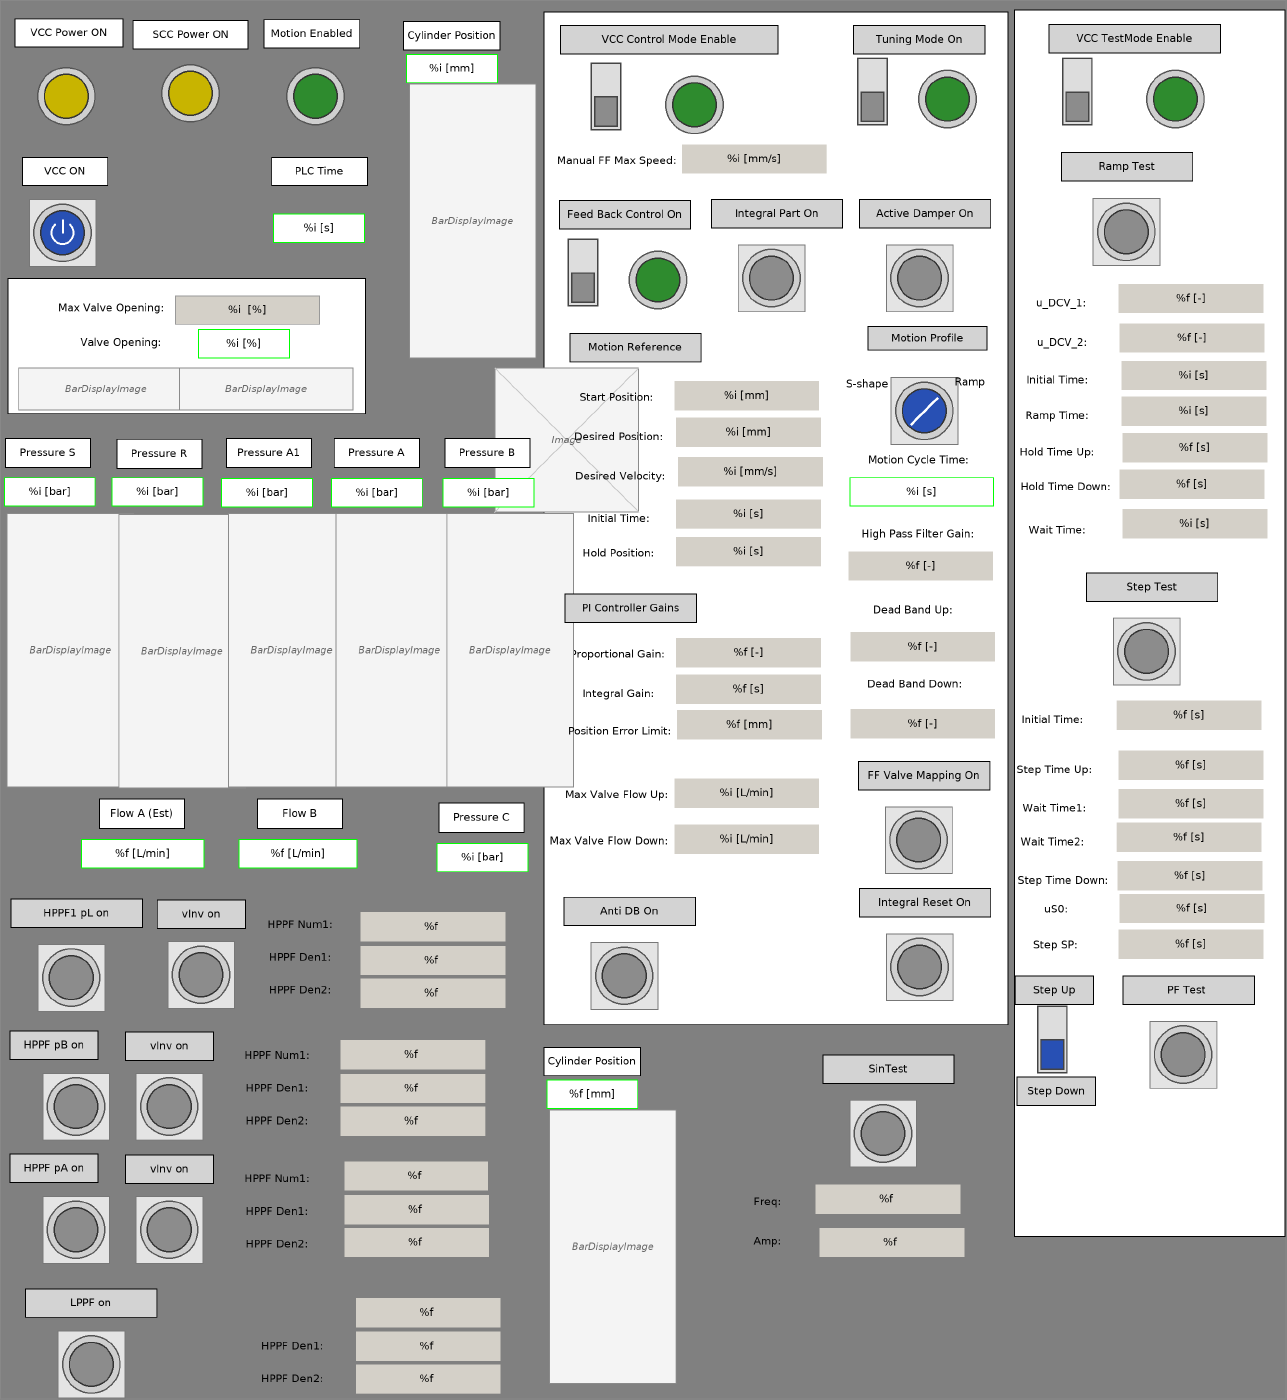
VISUALIZATION VCC_Visualization  // 1338x1455
    Rectangle (8,289 372x141)
    Rectangle (565,12 483x1053)
    Lamp1 (34,65 70x70), variable: GV.VCC_On_Light, style: Lamp-Lamp1-Yellow
    Lamp1 (163,62 70x70), variable: GV.SCC_On_Light, style: Lamp-Lamp1-Yellow
    Rectangle (23,163 89x30), "VCC ON"
    BarDisplayImage (425,87 132x285), value: UDP_Send.ActualCylPos, style: BarDisplayImage-Gray, scale format: %.1f, scale 0..500
        p518627256: mm
    Rectangle (15,19 113x30), "VCC Power ON"
    Rectangle (138,21 120x30), "SCC Power ON"
    Rectangle (419,22 101x30), "Cylinder Position"
    Image (514,382 150x150)
    DipSwitch (595,65 70x70), variable: GV.VCC_Control_Mode, behaviour: TOGGLE, style: Switch-DipSwitch-Gray
    Lamp1 (687,74 70x70), variable: VCC_Control_Mode_Enabled, style: Lamp-Lamp1-Green
    Rectangle (582,26 227x30), "VCC Control Mode Enable"
    Rectangle (581,208 137x30), "Feed Back Control On"
    Rectangle (739,207 137x30), "Integral Part On"
    PushSwitchLed (767,254 70x70), variable: VCC_I_Cntr_On, behaviour: TOGGLE, style: Switch-PushSwitchLed-Gray
    Label (568,439 150x30), "Desired Position:"
    Textfield (701,396 150x30), "%i [mm]", text variable: VCC_Cntrl_s0
        OnMouseClick: write the text variable via Default, min 0, max 500
    Label (566,398 150x30), "Start Position:"
    Textfield (703,434 150x30), "%i [mm]", text variable: VCC_Cntrl_Trvl_Dist
        OnMouseClick: write the text variable via Default, min 0, max 500-VCC_Cntrl_s0
    Textfield (705,475 150x30), "%i [mm/s]", text variable: VCC_Cntrl_Vel_SP
        OnMouseClick: write the text variable via Default, min 0, max 150
    Label (570,480 150x30), "Desired Velocity:"
    Label (874,619 150x30), "Dead Band Up:"
    Textfield (884,737 150x30), "%f [-]", text variable: VCC_Cntrl_DB_down
        OnMouseClick: write the text variable via Default, min 0.0000001, max 10.000000
    Textfield (703,519 150x30), "%i [s]", text variable: VCC_Cntrl_t0
        OnMouseClick: write the text variable via Default, min 0, max 20
    Label (568,524 150x30), "Initial Time:"
    Textfield (703,558 150x30), "%i [s]", text variable: VCC_Cntrl_tHold
        OnMouseClick: write the text variable via Default, min 0, max 20
    Label (568,560 150x30), "Hold Position:"
    Textfield (884,657 150x30), "%f [-]", text variable: VCC_Cntrl_DB_up
        OnMouseClick: write the text variable via Default, min 0, max 10
    Rectangle (1054,10 282x1275)
    DipSwitch (1085,60 70x70), variable: VCC_Test_Mode, behaviour: TOGGLE, style: Switch-DipSwitch-Gray
    Lamp1 (1187,68 70x70), variable: VCC_Test_Mode_Enabled, style: Lamp-Lamp1-Green
    Rectangle (1090,25 179x30), "VCC TestMode Enable"
    PushSwitchLed (1136,206 70x70), variable: VCC_Ramp_Test_On, behaviour: TOGGLE, style: Switch-PushSwitchLed-Gray
    Rectangle (1103,158 137x30), "Ramp Test"
    Textfield (1166,375 150x30), "%i [s]", text variable: VCC_Test_t0
        OnMouseClick: write the text variable via Default, min 0, max 500-VCC_Cntrl_s0
    Label (1024,380 150x30), "Initial Time:"
    Rectangle (855,1096 137x30), "SinTest"
    PushSwitchLed (883,1143 70x70), variable: VCC_Sin_Test_On, behaviour: TOGGLE, style: Switch-PushSwitchLed-Gray
    Label (567,665 150x30), "Proportional Gain:"
    Textfield (703,701 150x30), "%f [s]", text variable: VCC_Cntrl_T_I
        OnMouseClick: write the text variable via Default, min 0, max 1000
    Label (568,706 150x30), "Integral Gain:"
    Textfield (703,663 150x30), "%f [-]", text variable: VCC_Cntrl_k_P
        OnMouseClick: write the text variable via Default, min 0, max 100
    BarDisplayImage (7,533 132x285), value: UDP_Send.pP, style: BarDisplayImage-Gray, scale format: %.1f, scale 0..200
        p518627256: Bar
    Rectangle (5,455 89x31), "Pressure S"
    BarDisplayImage (123,534 132x285), value: UDP_Send.pR, style: BarDisplayImage-Gray, scale format: %.1f, scale 0..10
        p518627256: Bar
    Rectangle (121,456 89x31), "Pressure R"
    Rectangle (235,455 89x31), "Pressure A1"
    BarDisplayImage (237,533 132x285), value: UDP_Send.pA1, style: BarDisplayImage-Gray, scale format: %.1f, scale 0..200
        p518627256: Bar
    Rectangle (347,455 89x31), "Pressure A"
    BarDisplayImage (349,533 132x285), value: UDP_Send.pA, style: BarDisplayImage-Gray, scale format: %.1f, scale 0..200
        p518627256: Bar
    Rectangle (462,455 89x31), "Pressure B"
    BarDisplayImage (464,533 132x285), value: UDP_Send.pB, style: BarDisplayImage-Gray, scale format: %.1f, scale 0..200
        p518627256: Bar
    Textfield (422,56 95x30), "%i [mm]", text variable: UDP_Send.ActualCylPos
    Label (569,745 150x30), "Position Error Limit:"
    Textfield (704,738 150x30), "%f [mm]", text variable: VCC_Cntrl_Error_Limit
        OnMouseClick: write the text variable via Default, min 0, max 500-VCC_Cntrl_s0
    Lamp1 (293,65 70x70), variable: Motion_Start_Light, style: Lamp-Lamp1-Green
    Rectangle (274,20 100x30), "Motion Enabled"
    Label (566,152 150x30), "Manual FF Max Speed:"
    Textfield (709,150 150x30), "%i [mm/s]", text variable: VCC_Vel_Ref_Max
        OnMouseClick: write the text variable via Default, min 0, max 150
    Label (19,305 197x30), "Max Valve Opening:"
    Textfield (182,307 150x30), "%i [%]", text variable: VCC_Max_Joy_Output
        OnMouseClick: write the text variable via Default, min 0, max 100
    BarDisplayImage (19,382 182x44), value: UDP_Send.PVG_SP*100, style: BarDisplayImage-Gray, scale format: %.1f, scale -100..0
    BarDisplayImage (186,382 181x44), value: UDP_Send.PVG_SP*100, style: BarDisplayImage-Gray, scale format: %.1f, scale 0..100
    Rectangle (893,207 137x30), "Active Damper On"
    PushSwitchLed (921,254 70x70), variable: VCC_AD_On, behaviour: TOGGLE, style: Switch-PushSwitchLed-Gray
    Textfield (882,573 150x30), "%f [-]", text variable: VCC_k_AD
        OnMouseClick: write the text variable via Default, min 0, max 1
    Label (879,540 150x30), "High Pass Filter Gain:"
    DipSwitch (872,60 70x70), variable: VCC_Tuning_Mode, behaviour: TOGGLE, style: Switch-DipSwitch-Gray
    Rectangle (887,26 137x30), "Tuning Mode On"
    Lamp1 (950,68 70x70), variable: VCC_Tuning_Mode, style: Lamp-Lamp1-Green
    DipSwitch (571,248 70x70), variable: VCC_FB_Cntr_On, behaviour: TOGGLE, style: Switch-DipSwitch-Gray
    Lamp1 (649,256 70x70), variable: VCC_FB_Cntr_Enabled, style: Lamp-Lamp1-Green
    Label (876,696 150x30), "Dead Band Down:"
    Rectangle (587,617 137x30), "PI Controller Gains"
    Rectangle (592,346 137x30), "Motion Reference"
    RotarySwitch (926,392 70x70), variable: VCC_S_shape_On, behaviour: TOGGLE, style: Switch-RotarySwitch-Blue
    Rectangle (902,339 124x25), "Motion Profile"
    Label (975,382 67x30), "Ramp"
    Label (868,384 67x30), "S-shape"
    Rectangle (282,163 100x30), "PLC Time"
    Textfield (284,222 95x30), "%i [s]", text variable: UDP_Send.plcTime
    Label (880,463 150x30), "Motion Cycle Time:"
    Textfield (883,496 150x30), "%i [s]", text variable: VCC_Cntrl_Motion_Cycle_Time
    Label (566,811 150x30), "Max Valve Flow Up:"
    Textfield (701,809 150x30), "%i [L/min]", text variable: VCC_Cntrl_Q_max_up
        OnMouseClick: write the text variable via Default, min 0, max 70
    Label (29,341 197x30), "Valve Opening:"
    Textfield (206,342 95x30), "%i [%]", text variable: UDP_Send.PVG_SP*100
    Label (558,859 150x30), "Max Valve Flow Down:"
    Textfield (701,857 150x30), "%i [L/min]", text variable: VCC_Cntrl_Q_max_down
        OnMouseClick: write the text variable via Default, min 0, max 70
    Textfield (460,497 95x30), "%i [bar]", text variable: UDP_Send.pB
    Textfield (344,497 95x30), "%i [bar]", text variable: UDP_Send.pA
    Textfield (230,497 95x30), "%i [bar]", text variable: UDP_Send.pA1
    Textfield (116,496 95x30), "%i [bar]", text variable: UDP_Send.pR
    Textfield (4,496 95x30), "%i [bar]", text variable: UDP_Send.pP
    Rectangle (456,834 89x31), "Pressure C"
    Textfield (454,876 95x30), "%i [bar]", text variable: UDP_Send.pC
    Rectangle (103,830 89x31), "Flow A (Est)"
    Textfield (84,872 128x30), "%f [L/min]", text variable: abs(UDP_Send.QB*1.4083)
    Textfield (248,872 123x30), "%f [L/min]", text variable: abs(UDP_Send.QB)
    Rectangle (267,830 89x31), "Flow B"
    PushSwitchLed (920,838 70x70), variable: VCC_Cntrl_FF_Valve_Mapping_On, behaviour: TOGGLE, style: Switch-PushSwitchLed-Gray
    Rectangle (892,791 137x30), "FF Valve Mapping On"
    PushSwitchLed (921,970 70x70), variable: VCC_Cntrl_Integral_Reset_On, behaviour: TOGGLE, style: Switch-PushSwitchLed-Gray
    Rectangle (893,923 137x30), "Integral Reset On"
    PowerSwitch (30,207 70x70), variable: GV.VCC_ON, behaviour: TOGGLE, style: Switch-PowerSwitch-Blue
    Label (1028,300 150x30), "u_DCV_1:"
    Textfield (1163,295 150x30), "%f [-]", text variable: VCC_Ramp_Test_u_DCV_1
        OnMouseClick: write the text variable via Default, min -1, max 1
    Label (1029,341 150x30), "u_DCV_2:"
    Textfield (1164,336 150x30), "%f [-]", text variable: VCC_Ramp_Test_u_DCV_2
        OnMouseClick: write the text variable via Default, min -1, max 1
    Label (1024,417 150x30), "Ramp Time:"
    Textfield (1166,412 150x30), "%i [s]", text variable: VCC_Ramp_Test_tR
        OnMouseClick: write the text variable via Default, min 0, max 10
    Label (1024,455 150x30), "Hold Time Up:"
    Label (1024,536 150x30), "Wait Time:"
    Textfield (1167,450 150x30), "%f [s]", text variable: VCC_Ramp_Test_tHold_Up
        OnMouseClick: write the text variable via Default, min 0, max 10
    Textfield (1167,529 150x30), "%i [s]", text variable: VCC_Ramp_Test_tWait
        OnMouseClick: write the text variable via Default, min 0, max 10
    Label (1033,491 150x30), "Hold Time Down:"
    Textfield (1164,488 150x30), "%f [s]", text variable: VCC_Ramp_Test_tHold_Down
        OnMouseClick: write the text variable via Default, min 0, max 20
    PushSwitchLed (1157,642 70x70), variable: VCC_Step_Test_On, behaviour: TOGGLE, style: Switch-PushSwitchLed-Gray
    Rectangle (1129,595 137x30), "Step Test"
    Label (1019,733 150x30), "Initial Time:"
    Textfield (1161,728 150x30), "%f [s]", text variable: VCC_Step_Test_t0
        OnMouseClick: write the text variable via Default, min 0, max 500-VCC_Cntrl_s0
    Label (1021,785 150x30), "Step Time Up:"
    Textfield (1163,780 150x30), "%f [s]", text variable: VCC_Step_Test_tStepUp
        OnMouseClick: write the text variable via Default, min 0, max 500-VCC_Cntrl_s0
    Label (1023,930 150x30), "uS0:"
    Textfield (1164,929 150x30), "%f [s]", text variable: VCC_Step_Test_u0
        OnMouseClick: write the text variable via Default, min -1, max 1
    DipSwitch (1059,1045 70x70), variable: VCC_Step_Test_Up, behaviour: TOGGLE, style: Switch-DipSwitch-Blue
    Rectangle (1057,1119 82x30), "Step Down"
    Rectangle (1055,1014 82x30), "Step Up"
    Label (1021,825 150x30), "Wait Time1:"
    Textfield (1163,820 150x30), "%f [s]", text variable: VCC_Step_Test_tWait
        OnMouseClick: write the text variable via Default, min 0, max 500-VCC_Cntrl_s0
    Label (1030,900 150x30), "Step Time Down:"
    Textfield (1162,895 150x30), "%f [s]", text variable: VCC_Step_Test_tStepDown
        OnMouseClick: write the text variable via Default, min 0, max 500-VCC_Cntrl_s0
    Label (1019,860 150x30), "Wait Time2:"
    Textfield (1161,855 150x30), "%f [s]", text variable: VCC_Step_Test_tWait2
        OnMouseClick: write the text variable via Default, min 0, max 500-VCC_Cntrl_s0
    Label (1022,967 150x30), "Step SP:"
    Textfield (1163,966 150x30), "%f [s]", text variable: VCC_Step_Test_SP
        OnMouseClick: write the text variable via Default, min -1, max 1
    Label (237,946 150x30), "HPPF Num1:"
    Textfield (375,948 150x30), "%f", text variable: VCC_PF1_HP_Num1
        OnMouseClick: write the text variable via Default, min -1.000000000000000000000000000000000000000001, max 1.000000000000000000000000000000000000000000000000001
    Label (141,984 150x30)
    Label (237,980 150x30), "HPPF Den1:"
    Textfield (375,983 150x30), "%f", text variable: VCC_PF1_HP_Den1
        OnMouseClick: write the text variable via Default, min -1, max 1
    Label (237,1014 150x30), "HPPF Den2:"
    Textfield (375,1017 150x30), "%f", text variable: VCC_PF1_HP_Den2
        OnMouseClick: write the text variable via Default, min -1, max 1
    Rectangle (1167,1014 137x30), "PF Test"
    PushSwitchLed (1195,1061 70x70), variable: VCC_PF_Test_On, behaviour: TOGGLE, style: Switch-PushSwitchLed-Gray
    PushSwitchLed (39,981 70x70), variable: VCC_PF1_On, behaviour: TOGGLE, style: Switch-PushSwitchLed-Gray
    Rectangle (11,934 137x30), "HPPF1 pL on"
    PushSwitchLed (614,979 70x70), variable: VCC_PF_ADB_On, behaviour: TOGGLE, style: Switch-PushSwitchLed-Gray
    Rectangle (586,932 137x30), "Anti DB On"
    Label (723,964 150x30)
    PushSwitchLed (60,1383 70x70), variable: VCC_LPPF_On, behaviour: TOGGLE, style: Switch-PushSwitchLed-Gray
    Rectangle (26,1339 137x30), "LPPF on"
    Label (723,1234 150x30), "Freq:"
    Textfield (370,1349 150x30), "%f", text variable: VCC_LPPF_Num1
        OnMouseClick: write the text variable via Default, min -1.000000000000000000000000000000000000000001, max 1.000000000000000000000000000000000000000000000000001
    Label (229,1384 150x30), "HPPF Den1:"
    Textfield (370,1384 150x30), "%f", text variable: VCC_LPPF_Den1
        OnMouseClick: write the text variable via Default, min -1, max 1
    Label (229,1418 150x30), "HPPF Den2:"
    Textfield (370,1418 150x30), "%f", text variable: VCC_LPPF_Den2
        OnMouseClick: write the text variable via Default, min -1, max 1
    PushSwitchLed (44,1115 70x70), variable: VCC_PF_pB_On, behaviour: TOGGLE, style: Switch-PushSwitchLed-Gray
    Rectangle (10,1071 92x30), "HPPF pB on"
    Label (213,1082 150x30), "HPPF Num1:"
    Textfield (354,1081 150x30), "%f", text variable: VCC_PF_pB_HP_Num1
        OnMouseClick: write the text variable via Default, min -1.000000000000000000000000000000000000000001, max 1.000000000000000000000000000000000000000000000000001
    Label (213,1116 150x30), "HPPF Den1:"
    Textfield (354,1116 150x30), "%f", text variable: VCC_PF_pB_HP_Den1
        OnMouseClick: write the text variable via Default, min -1, max 1
    Label (213,1150 150x30), "HPPF Den2:"
    Textfield (354,1150 150x30), "%f", text variable: VCC_PF_pB_HP_Den2
        OnMouseClick: write the text variable via Default, min -1, max 1
    BarDisplayImage (571,1153 132x285), value: UDP_Send.ActualCylPos, style: BarDisplayImage-Gray, scale format: %.1f, scale 0..500
        p518627256: mm
    Rectangle (565,1088 101x30), "Cylinder Position"
    Textfield (568,1122 95x30), "%f [mm]", text variable: UDP_Send.ActualCylPos
    PushSwitchLed (141,1115 70x70), variable: VCC_PF_pB_vInv_On, behaviour: TOGGLE, style: Switch-PushSwitchLed-Gray
    Rectangle (130,1072 92x30), "vInv on"
    PushSwitchLed (174,978 70x70), variable: VCC_PF_pL_vInv_On, behaviour: TOGGLE, style: Switch-PushSwitchLed-Gray
    Rectangle (163,935 92x30), "vInv on"
    Textfield (848,1231 150x30), "%f", text variable: VCC_SinTest_freq
        OnMouseClick: write the text variable via Default, min -1.000000000000000000000000000000000000000001, max 1.000000000000000000000000000000000000000000000000001
    Textfield (852,1276 150x30), "%f", text variable: VCC_SinTest_Amp
        OnMouseClick: write the text variable via Default, min -1.000000000000000000000000000000000000000001, max 1.000000000000000000000000000000000000000000000000001
    Label (723,1275 150x30), "Amp:"
    PushSwitchLed (44,1243 70x70), variable: VCC_PF2_On, behaviour: TOGGLE, style: Switch-PushSwitchLed-Gray
    Rectangle (10,1199 92x30), "HPPF pA on"
    Label (213,1210 150x30), "HPPF Num1:"
    Label (213,1244 150x30), "HPPF Den1:"
    Label (213,1278 150x30), "HPPF Den2:"
    PushSwitchLed (141,1243 70x70), variable: VCC_PF_pA_vInv_On, behaviour: TOGGLE, style: Switch-PushSwitchLed-Gray
    Rectangle (130,1200 92x30), "vInv on"
    Textfield (358,1207 149x30), "%f", text variable: VCC_PF_HP_Num1
        OnMouseClick: write the text variable via Default, min -1.000000000000000000000000000000000000000001, max 1.000000000000000000000000000000000000000000000000001
    Textfield (358,1242 150x30), "%f", text variable: VCC_PF_HP_Den1
        OnMouseClick: write the text variable via Default, min -1, max 1
    Textfield (358,1276 150x30), "%f", text variable: VCC_PF_HP_Den2
        OnMouseClick: write the text variable via Default, min -1, max 1
END_VISUALIZATION

// IndraMotionMlc1/Application/Visualization/SCC/SubWindows/SCC_Main
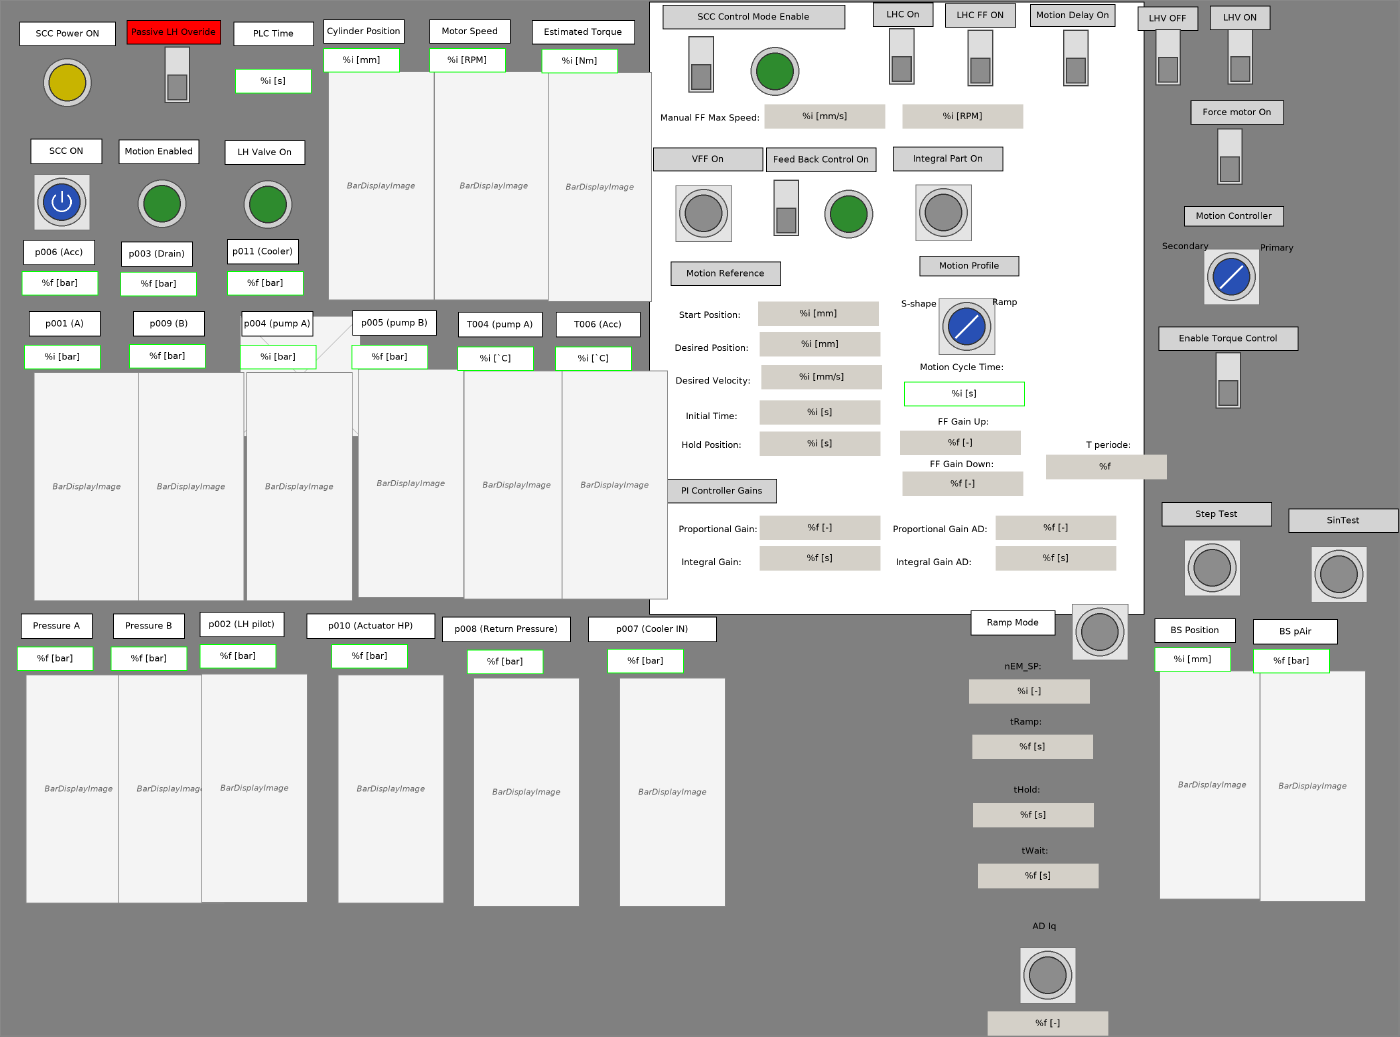
VISUALIZATION SCC_Main  // 1745x1293
    Lamp1 (49,68 70x70), variable: GV.SCC_On_Light, style: Lamp-Lamp1-Yellow
    Rectangle (38,173 89x31), "SCC ON"
    BarDisplayImage (409,89 132x285), value: UDP_Send.ActualCylPos, style: BarDisplayImage-Gray, scale format: %.1f, scale 0..500
        p518627256: mm
    Rectangle (24,27 120x30), "SCC Power ON"
    Rectangle (403,24 101x30), "Cylinder Position"
    Image (299,394 150x150)
    Rectangle (29,299 89x31), "p006 (Acc)"
    Rectangle (26,765 89x31), "Pressure A"
    BarDisplayImage (32,841 132x285), value: UDP_Send.pA, style: BarDisplayImage-Gray, scale format: %.1f, scale 0..160
        p518627256: Bar
    Rectangle (141,765 89x31), "Pressure B"
    BarDisplayImage (147,841 132x285), value: UDP_Send.pB, style: BarDisplayImage-Gray, scale format: %.1f, scale 0..160
        p518627256: Bar
    Lamp1 (167,219 70x70), variable: Motion_Start_Light, style: Lamp-Lamp1-Green
    Rectangle (148,174 100x30), "Motion Enabled"
    Rectangle (36,388 89x31), "p001 (A)"
    BarDisplayImage (42,464 132x285), value: UDP_Send.p_001, style: BarDisplayImage-Gray, scale format: %.1f, scale 0..160
        p518627256: Bar
    Rectangle (166,388 89x31), "p009 (B)"
    BarDisplayImage (172,464 132x285), value: UDP_Send.p_009, style: BarDisplayImage-Gray, scale format: %.1f, scale 0..160
        p518627256: Bar
    Rectangle (301,388 89x31), "p004 (pump A)"
    BarDisplayImage (307,464 132x285), value: UDP_Send.p_004, style: BarDisplayImage-Gray, scale format: %.1f, scale 0..160
        p518627256: Bar
    Rectangle (439,387 105x31), "p005 (pump B)"
    BarDisplayImage (446,460 132x285), value: UDP_Send.p_005, style: BarDisplayImage-Gray, scale format: %.1f, scale 0..160
        p518627256: Bar
    Rectangle (283,298 89x31), "p011 (Cooler)"
    Rectangle (151,301 89x31), "p003 (Drain)"
    Rectangle (249,763 105x31), "p002 (LH pilot)"
    BarDisplayImage (251,840 132x285), value: UDP_Send.p_002, style: BarDisplayImage-Gray, scale format: %.1f, scale 0..160
        p518627256: Bar
    Rectangle (382,765 160x31), "p010 (Actuator HP)"
    BarDisplayImage (421,841 132x285), value: UDP_Send.p_010, style: BarDisplayImage-Gray, scale format: %.1f, scale 0..160
        p518627256: Bar
    BarDisplayImage (590,845 132x285), value: UDP_Send.p_008, style: BarDisplayImage-Gray, scale format: %.1f, scale 0..160
        p518627256: Bar
    Rectangle (551,769 160x31), "p008 (Return Pressure)"
    BarDisplayImage (772,845 132x285), value: UDP_Send.p_007, style: BarDisplayImage-Gray, scale format: %.1f, scale 0..160
        p518627256: Bar
    Rectangle (733,769 160x31), "p007 (Cooler IN)"
    Textfield (403,60 95x30), "%i [mm]", text variable: UDP_Send.ActualCylPos
    Textfield (27,338 95x30), "%f [bar]", text variable: UDP_Send.p_006
    Textfield (150,339 95x30), "%f [bar]", text variable: UDP_Send.p_003
    Textfield (283,338 95x30), "%f [bar]", text variable: UDP_Send.p_011
    Textfield (21,806 95x30), "%f [bar]", text variable: UDP_Send.pA
    Textfield (138,806 95x30), "%f [bar]", text variable: UDP_Send.pB
    Textfield (30,430 95x30), "%i [bar]", text variable: UDP_Send.p_001
    Textfield (161,429 95x30), "%f [bar]", text variable: UDP_Send.p_009
    Textfield (299,430 95x30), "%i [bar]", text variable: UDP_Send.p_004
    Textfield (438,430 95x30), "%f [bar]", text variable: UDP_Send.p_005
    Textfield (249,803 95x30), "%f [bar]", text variable: UDP_Send.p_002
    Textfield (413,803 95x30), "%f [bar]", text variable: UDP_Send.p_010
    Textfield (582,810 95x30), "%f [bar]", text variable: UDP_Send.p_008
    Textfield (757,809 95x30), "%f [bar]", text variable: UDP_Send.p_007
    Rectangle (535,24 101x30), "Motor Speed"
    BarDisplayImage (541,89 149x285), value: abs(UDP_Send.ActualVel), style: BarDisplayImage-Gray, scale format: %.1f, scale 0..3500
        p518627256: mm
    Textfield (535,60 95x30), "%i [RPM]", text variable: UDP_Send.ActualVel
    Rectangle (291,27 100x30), "PLC Time"
    Textfield (293,86 95x30), "%i [s]", text variable: UDP_Send.plcTime
    Rectangle (809,2 617x764)
    DipSwitch (839,45 70x70), variable: SCC_Control_Mode, behaviour: TOGGLE, style: Switch-DipSwitch-Gray
    Lamp1 (931,54 70x70), variable: SCC_Control_Mode_Enabled, style: Lamp-Lamp1-Green
    Rectangle (826,6 227x30), "SCC Control Mode Enable"
    Rectangle (955,184 137x30), "Feed Back Control On"
    Rectangle (1113,183 137x30), "Integral Part On"
    PushSwitchLed (1141,230 70x70), variable: SCC_I_Cntr_On, behaviour: TOGGLE, style: Switch-PushSwitchLed-Gray
    Label (812,419 150x30), "Desired Position:"
    Textfield (945,376 150x30), "%i [mm]", text variable: SCC_Cntrl_s0
        OnMouseClick: write the text variable via Default, min 0, max 500
    Label (810,378 150x30), "Start Position:"
    Textfield (947,414 150x30), "%i [mm]", text variable: SCC_Cntrl_Pos_SP
        OnMouseClick: write the text variable via Default, min 0, max 490
    Textfield (949,455 150x30), "%i [mm/s]", text variable: SCC_Cntrl_Vel_SP
        OnMouseClick: write the text variable via Default, min 0, max 150
    Label (814,460 150x30), "Desired Velocity:"
    Textfield (947,499 150x30), "%i [s]", text variable: SCC_Cntrl_t0
        OnMouseClick: write the text variable via Default, min 0, max 20
    Label (812,504 150x30), "Initial Time:"
    Textfield (947,538 150x30), "%i [s]", text variable: SCC_Cntrl_tHold_Up_Up_Up
        OnMouseClick: write the text variable via Default, min 0, max 20
    Label (812,540 150x30), "Hold Position:"
    Label (820,645 150x30), "Proportional Gain:"
    Textfield (947,681 150x30), "%f [s]", text variable: SCC_Cntrl_T_I
        OnMouseClick: write the text variable via Default, min 0, max 1e10
    Label (812,686 150x30), "Integral Gain:"
    Textfield (947,643 150x30), "%f [-]", text variable: SCC_Cntrl_k_P
        OnMouseClick: write the text variable via Default, min 0, max 1e10
    Label (810,132 150x30), "Manual FF Max Speed:"
    Textfield (953,130 150x30), "%i [mm/s]", text variable: SCC_Vel_Ref_Max
        OnMouseClick: write the text variable via Default, min 0, max 150
    DipSwitch (1306,37 70x70), variable: SCC_Motion_Delay_On, behaviour: TOGGLE, style: Switch-DipSwitch-Gray
    Rectangle (1284,5 106x28), "Motion Delay On"
    DipSwitch (945,224 70x70), variable: SCC_FB_Cntr_On, behaviour: TOGGLE, style: Switch-DipSwitch-Gray
    Lamp1 (1023,232 70x70), variable: SCC_FB_Cntr_Enabled, style: Lamp-Lamp1-Green
    Rectangle (831,597 137x30), "PI Controller Gains"
    Rectangle (836,326 137x30), "Motion Reference"
    RotarySwitch (1170,372 70x70), variable: SCC_S_shape_On, behaviour: TOGGLE, style: Switch-RotarySwitch-Blue
    Rectangle (1146,319 124x25), "Motion Profile"
    Label (1219,362 67x30), "Ramp"
    Label (1112,364 67x30), "S-shape"
    Label (1124,443 150x30), "Motion Cycle Time:"
    Textfield (1127,476 150x30), "%i [s]", text variable: SCC_Cntrl_Motion_Cycle_Time
    Textfield (1125,130 150x30), "%i [RPM]", text variable: SCC_Manual_Max_Speed
        OnMouseClick: write the text variable via Default, min 0, max 3500
    Lamp1 (299,220 70x70), variable: SCC_LH_Valve_Activated, style: Lamp-Lamp1-Green
    Rectangle (280,175 100x30), "LH Valve On"
    BarDisplayImage (578,462 132x285), value: UDP_Send.T004, style: BarDisplayImage-Gray, scale format: %.1f, scale 0..50
        p518627256: Bar
    Rectangle (571,389 105x31), "T004 (pump A)"
    Textfield (570,432 95x30), "%i [`C]", text variable: UDP_Send.T004
    BarDisplayImage (700,462 132x285), value: UDP_Send.T006, style: BarDisplayImage-Gray, scale format: %.1f, scale 0..50
        p518627256: Bar
    Rectangle (693,389 105x31), "T006 (Acc)"
    Textfield (692,432 95x30), "%i [`C]", text variable: UDP_Send.T006
    Textfield (1122,537 150x30), "%f [-]", text variable: SCC_Cntrl_FF_up
        OnMouseClick: write the text variable via Default, min 0, max 1e10
    Label (1126,511 150x30), "FF Gain Up:"
    Textfield (1125,588 150x30), "%f [-]", text variable: SCC_Cntrl_FF_down
        OnMouseClick: write the text variable via Default, min 0, max 1e10
    Label (1124,564 150x30), "FF Gain Down:"
    BarDisplayImage (683,90 129x286), value: abs(UDP_Send.Sc_DataC)*2.05, style: BarDisplayImage-Gray, scale format: %.1f, scale -50..50
        p518627256: mm
    Rectangle (663,25 128x30), "Estimated Torque"
    Textfield (675,61 95x30), "%i [Nm]", text variable: abs(UDP_Send.Sc_DataC)*2.05
    DipSwitch (186,58 70x70), variable: TestMode, behaviour: TOGGLE, style: Switch-DipSwitch-Gray
    Rectangle (158,25 117x30), "Passive LH Overide"
    Label (1200,816 150x30), "nEM_SP:"
    Textfield (1208,847 150x30), "%i [-]", text variable: nSP
        OnMouseClick: write the text variable via Default, min -4200, max 4200
    Label (1204,885 150x30), "tRamp:"
    Textfield (1212,916 150x30), "%f [s]", text variable: tRamp
        OnMouseClick: write the text variable via Default, min 0, max 100
    Label (1205,970 150x30), "tHold:"
    Textfield (1213,1001 150x30), "%f [s]", text variable: Ramp_tHold
        OnMouseClick: write the text variable via Default, min 0, max 100
    Label (1215,1046 150x30), "tWait:"
    Textfield (1219,1077 150x30), "%f [s]", text variable: Ramp_tWait
        OnMouseClick: write the text variable via Default, min 0, max 100
    Rectangle (1210,761 105x31), "Ramp Mode"
    Rectangle (814,184 137x29), "VFF On"
    PushSwitchLed (842,231 70x70), variable: SCC_Cntrl_FF_On, behaviour: TOGGLE, style: Switch-PushSwitchLed-Gray
    PushSwitchLed (1336,753 70x70), variable: SCC_OL_On, behaviour: TOGGLE, style: Switch-PushSwitchLed-Gray
    Rectangle (1606,634 137x30), "SinTest"
    PushSwitchLed (1634,681 70x70), variable: SCC_Sin_Test_On, behaviour: TOGGLE, style: Switch-PushSwitchLed-Gray
    Label (1307,540 150x30), "T periode:"
    Textfield (1304,567 150x30), "%f", text variable: SCC_SinTest_T
        OnMouseClick: write the text variable via Default, min -1.000000000000000000000000000000000000000001, max 1.000000000000000000000000000000000000000000000000001
    DipSwitch (1089,35 70x70), variable: SCC_LHC_On, behaviour: TOGGLE, style: Switch-DipSwitch-Gray
    Rectangle (1088,3 75x30), "LHC On"
    Textfield (1241,643 150x30), "%f [-]", text variable: SCC_Cntrl_k_P_AD
        OnMouseClick: write the text variable via Default, min 0, max 1e10
    Label (1097,645 150x30), "Proportional Gain AD:"
    Textfield (1241,681 150x30), "%f [s]", text variable: SCC_Cntrl_T_I_AD
        OnMouseClick: write the text variable via Default, min 0, max 1e10
    Label (1089,686 150x30), "Integral Gain AD:"
    Rectangle (1418,8 75x30), "LHV OFF"
    DipSwitch (1421,36 70x70), variable: SCC_LHV_OFF, behaviour: TOGGLE, style: Switch-DipSwitch-Gray
    PushSwitchLed (1476,673 70x70), variable: SCC_Step_Test_On, behaviour: TOGGLE, style: Switch-PushSwitchLed-Gray
    Rectangle (1448,626 137x30), "Step Test"
    PowerSwitch (42,217 70x70), variable: GV.SCC_ON, behaviour: TOGGLE, style: Switch-PowerSwitch-Blue
    DipSwitch (1511,35 70x70), variable: SCC_LHV_ON, behaviour: TOGGLE, style: Switch-DipSwitch-Gray
    Rectangle (1508,7 75x30), "LHV ON"
    DipSwitch (1498,160 70x70), variable: SCC_Force_Motor_ON, behaviour: TOGGLE, style: Switch-DipSwitch-Gray
    Rectangle (1484,125 116x30), "Force motor On"
    DipSwitch (1187,37 70x70), variable: SCC_LHC_FF_On, behaviour: TOGGLE, style: Switch-DipSwitch-Gray
    Rectangle (1178,4 88x30), "LHC FF ON"
    Label (1227,1140 150x30), "AD Iq"
    PushSwitchLed (1271,1181 70x70), variable: SCC_AD_Iq_On, behaviour: TOGGLE, style: Switch-PushSwitchLed-Gray
    Textfield (1231,1261 150x30), "%f [-]", text variable: SCC_k_AD_Iq
        OnMouseClick: write the text variable via Default, min 0, max 1e15
    BarDisplayImage (1445,836 132x285), value: UDP_Send.T011, style: BarDisplayImage-Gray, scale format: %.1f, scale 0..150
        p518627256: mm
    Rectangle (1439,771 101x30), "BS Position"
    Textfield (1439,807 95x30), "%i [mm]", text variable: UDP_Send.T011
    BarDisplayImage (1570,836 132x288), value: UDP_Send.T004, style: BarDisplayImage-Gray, scale format: %.1f, scale 0..10
        p518627256: Bar
    Rectangle (1562,772 105x31), "BS pAir"
    Textfield (1562,809 95x30), "%f [bar]", text variable: UDP_Send.T004
    Label (1558,294 67x30), "Primary"
    RotarySwitch (1500,310 70x70), variable: SCC_SCTR_ON, behaviour: TOGGLE, style: Switch-RotarySwitch-Blue
    Rectangle (1476,257 124x25), "Motion Controller"
    Label (1444,292 67x30), "Secondary"
    DipSwitch (1496,439 70x70), variable: SCC_Enable_TCTR, behaviour: TOGGLE, style: Switch-DipSwitch-Gray
    Rectangle (1444,407 174x30), "Enable Torque Control"
END_VISUALIZATION

// IndraMotionMlc1/Application/Visualization/VCC/VCC_Filtered_LS
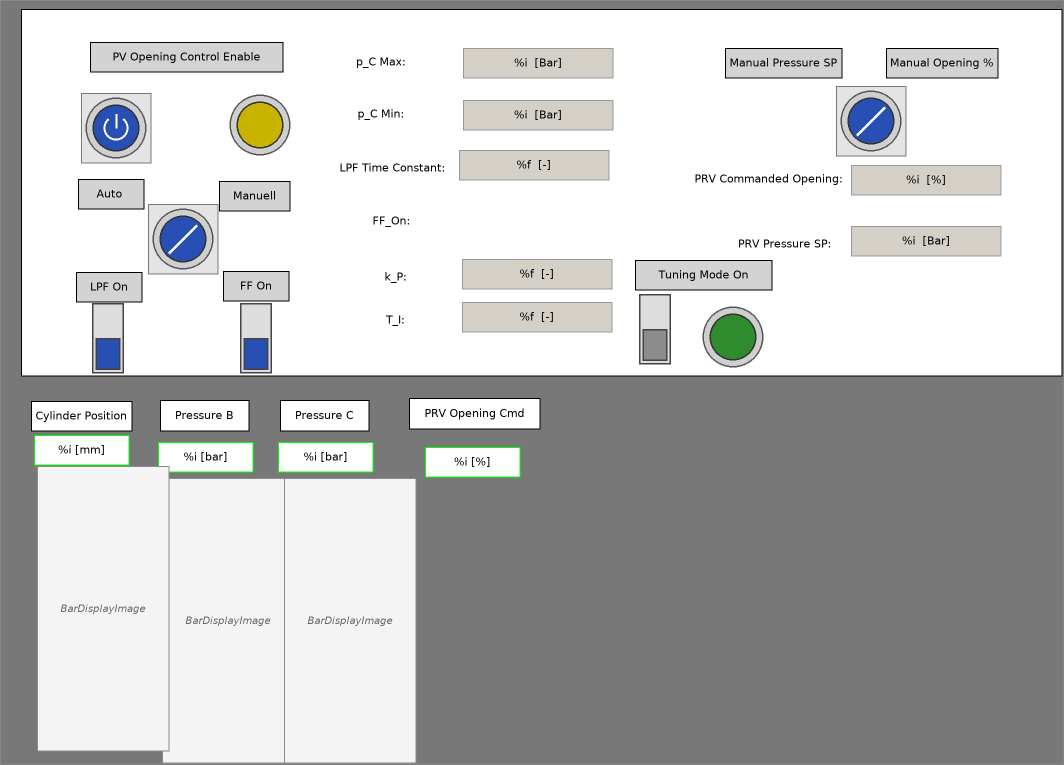
VISUALIZATION VCC_Filtered_LS  // 1064x765
    Rectangle (21,9 1041x367)
    Rectangle (78,179 66x30), "Auto"
    Textfield (463,48 150x30), "%i [Bar]", text variable: VCC_PRV_Cntrl_p_C_Max
        OnMouseClick: write the text variable via Default, min 0, max 100
    Label (284,47 197x30), "p_C Max:"
    Textfield (425,447 95x30), "%i [%]", text variable: UDP_Send.PRV_Cmd_Opening*100
    Label (284,99 197x30), "p_C Min:"
    Textfield (463,100 150x30), "%i [Bar]", text variable: VCC_PRV_Cntrl_p_C_Min
        OnMouseClick: write the text variable via Default, min 0, max 100
    Textfield (851,165 150x30), "%i [%]", text variable: VCC_PRV_Cntrl_Opening_SP
        OnMouseClick: write the text variable via Default, min 0, max 100
    Label (672,164 197x30), "PRV Commanded Opening:"
    RotarySwitch (836,86 70x70), variable: VCC_PRV_Cntrl_Manual_Pressure_On, behaviour: TOGGLE, style: Switch-RotarySwitch-Blue
    Rectangle (886,48 112x30), "Manual Opening %"
    Rectangle (725,48 117x30), "Manual Pressure SP"
    Label (686,229 197x30), "PRV Pressure SP:"
    Textfield (851,226 150x30), "%i [Bar]", text variable: VCC_PRV_p_C_SP
        OnMouseClick: write the text variable via Default, min 0, max 100
    Rectangle (160,400 89x31), "Pressure B"
    BarDisplayImage (162,478 132x285), value: UDP_Send.pB, style: BarDisplayImage-Gray, scale format: %.1f, scale 0..200
        p518627256: Bar
    Textfield (158,442 95x30), "%i [bar]", text variable: UDP_Send.pB
    Rectangle (280,400 89x31), "Pressure C"
    Textfield (278,442 95x30), "%i [bar]", text variable: UDP_Send.pC
    BarDisplayImage (284,478 132x285), value: UDP_Send.pC, style: BarDisplayImage-Gray, scale format: %.1f, scale 0..200
        p518627256: Bar
    Label (294,153 197x30), "LPF Time Constant:"
    Textfield (459,150 150x30), "%f [-]", text variable: VCC_PRV_Cntrl_T_LPF
        OnMouseClick: write the text variable via Default, min 0, max 100
    RotarySwitch (148,204 70x70), variable: VCC_PRV_Cntrl_Auto_On, behaviour: TOGGLE, style: Switch-RotarySwitch-Blue
    Rectangle (219,181 71x30), "Manuell"
    Rectangle (90,42 193x30), "PV Opening Control Enable"
    PowerSwitch (81,93 70x70), variable: VCC_PRV_Cntrl_Enable, behaviour: TOGGLE, style: Switch-PowerSwitch-Blue
    Lamp1 (225,90 70x70), variable: VCC_PRV_Cntrl_Enabled, style: Lamp-Lamp1-Yellow
    Label (297,262 197x30), "k_P:"
    Textfield (462,259 150x30), "%f [-]", text variable: VCC_PRV_Cntrl_k_P
        OnMouseClick: write the text variable via Default, min 0, max 100
    Label (297,305 197x30), "T_I:"
    Textfield (462,302 150x30), "%f [-]", text variable: VCC_PRV_Cntrl_T_I
        OnMouseClick: write the text variable via Default, min 0, max 100
    Label (293,206 197x30), "FF_On:"
    DipSwitch (221,303 70x70), variable: VCC_PRV_Cntrl_FF_On, behaviour: TOGGLE, style: Switch-DipSwitch-Blue
    Rectangle (409,398 131x31), "PRV Opening Cmd"
    Rectangle (223,271 66x30), "FF On"
    DipSwitch (73,303 70x70), variable: VCC_PRV_Cntrl_LPF_On, behaviour: TOGGLE, style: Switch-DipSwitch-Blue
    Rectangle (76,272 66x30), "LPF On"
    Rectangle (31,401 101x30), "Cylinder Position"
    BarDisplayImage (37,466 132x285), value: UDP_Send.ActualCylPos, style: BarDisplayImage-Gray, scale format: %.1f, scale 0..500
        p518627256: mm
    Textfield (34,435 95x30), "%i [mm]", text variable: UDP_Send.ActualCylPos
    DipSwitch (620,294 70x70), variable: VCC_PRV_Cntrl_Tuning_Mode_On, behaviour: TOGGLE, style: Switch-DipSwitch-Gray
    Rectangle (635,260 137x30), "Tuning Mode On"
    Lamp1 (698,302 70x70), variable: VCC_PRV_Cntrl_Tuning_Mode_On, style: Lamp-Lamp1-Green
END_VISUALIZATION

// IndraMotionMlc1/Application/Visualization/SCC/SubWindows/SCC_activeDamping
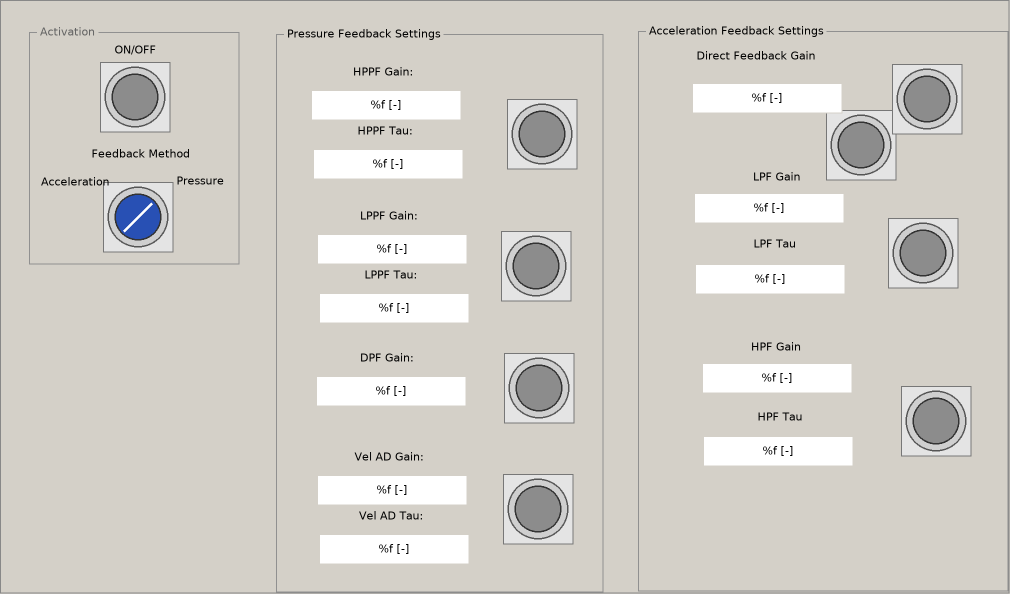
VISUALIZATION SCC_activeDamping  // 1010x594
    GroupBox (29,24 210x240), "Activation"
        RotarySwitch (74,158 70x70), variable: SCC_AF_On, behaviour: TOGGLE, style: Switch-RotarySwitch-Blue
        Label (13,143 67x30), "Acceleration"
        PushSwitchLed (71,38 70x70), variable: SCC_AD_On, behaviour: TOGGLE, style: Switch-PushSwitchLed-Gray
        Label (138,142 67x30), "Pressure"
        Label (73,11 67x30), "ON/OFF"
        Label (36,115 152x30), "Feedback Method"
    GroupBox (276,26 327x566), "Pressure Feedback Settings"
        Textfield (35,64 150x30), "%f [-]", text variable: SCC_HPPF_kf
            OnMouseClick: write the text variable via Default, min 0, max 100
        Label (32,31 150x30), "HPPF Gain:"
        Label (34,90 150x30), "HPPF Tau:"
        Textfield (37,123 150x30), "%f [-]", text variable: SCC_HPPF_tauf
            OnMouseClick: write the text variable via Default, min 0, max 100
        Textfield (41,208 150x30), "%f [-]", text variable: SCC_LPPF_kf
            OnMouseClick: write the text variable via Default, min 0, max 100
        Label (38,175 150x30), "LPPF Gain:"
        Label (40,234 150x30), "LPPF Tau:"
        Textfield (43,267 150x30), "%f [-]", text variable: SCC_LPPF_tauf
            OnMouseClick: write the text variable via Default, min 0, max 100
        Label (36,317 150x30), "DPF Gain:"
        PushSwitchLed (225,205 70x70), variable: SCC_LPPF_On, behaviour: TOGGLE, style: Switch-PushSwitchLed-Gray
        PushSwitchLed (228,327 70x70), variable: SCC_DPF_On, behaviour: TOGGLE, style: Switch-PushSwitchLed-Gray
        Textfield (41,449 150x30), "%f [-]", text variable: SCC_vel_AD_kf
            OnMouseClick: write the text variable via Default, min 0, max 1000000
        Label (38,416 150x30), "Vel AD Gain:"
        Label (40,475 150x30), "Vel AD Tau:"
        Textfield (43,508 150x30), "%f [-]", text variable: SCC_vel_AD_tauf
            OnMouseClick: write the text variable via Default, min 0, max 100
        PushSwitchLed (227,448 70x70), variable: SCC_vel_AD_On, behaviour: TOGGLE, style: Switch-PushSwitchLed-Gray
        PushSwitchLed (550,84 70x70), variable: SCC_HPPF_On, behaviour: TOGGLE, style: Switch-PushSwitchLed-Gray
        PushSwitchLed (231,73 70x70), variable: SCC_HPPF_On, behaviour: TOGGLE, style: Switch-PushSwitchLed-Gray
        Textfield (40,350 150x30), "%f [-]", text variable: SCC_DPF_kf
            OnMouseClick: write the text variable via Default, min 0, max 100
        Label (38,376 150x30)
    GroupBox (638,23 370x568), "Acceleration Feedback Settings"
        PushSwitchLed (263,363 70x70), variable: SCC_AF_HPF_On, behaviour: TOGGLE, style: Switch-PushSwitchLed-Gray
        PushSwitchLed (254,41 70x70), variable: SCC_AF_Direct_On, behaviour: TOGGLE, style: Switch-PushSwitchLed-Gray
        PushSwitchLed (250,195 70x70), variable: SCC_AF_LPF_On, behaviour: TOGGLE, style: Switch-PushSwitchLed-Gray
        Textfield (54,60 150x30), "%f [-]", text variable: SCC_AF_K_direct
            OnMouseClick: write the text variable via Default
        Label (43,18 150x30), "Direct Feedback Gain"
        Label (67,379 150x30), "HPF Tau"
        Label (63,309 150x30), "HPF Gain"
        Label (62,206 150x30), "LPF Tau"
        Label (64,139 150x30), "LPF Gain"
        Textfield (56,170 150x30), "%f [-]", text variable: SCC_AF_LPF_Num2
            OnMouseClick: write the text variable via Default
        Textfield (57,241 150x30), "%f [-]", text variable: SCC_AF_LPF_Den2
            OnMouseClick: write the text variable via Default
        Textfield (64,340 150x30), "%f [-]", text variable: SCC_AF_HPF_Num1
            OnMouseClick: write the text variable via Default
        Textfield (65,413 150x30), "%f [-]", text variable: SCC_AF_HPF_Den2
            OnMouseClick: write the text variable via Default
END_VISUALIZATION

// IndraMotionMlc1/Application/Visualization/SCC/SCC
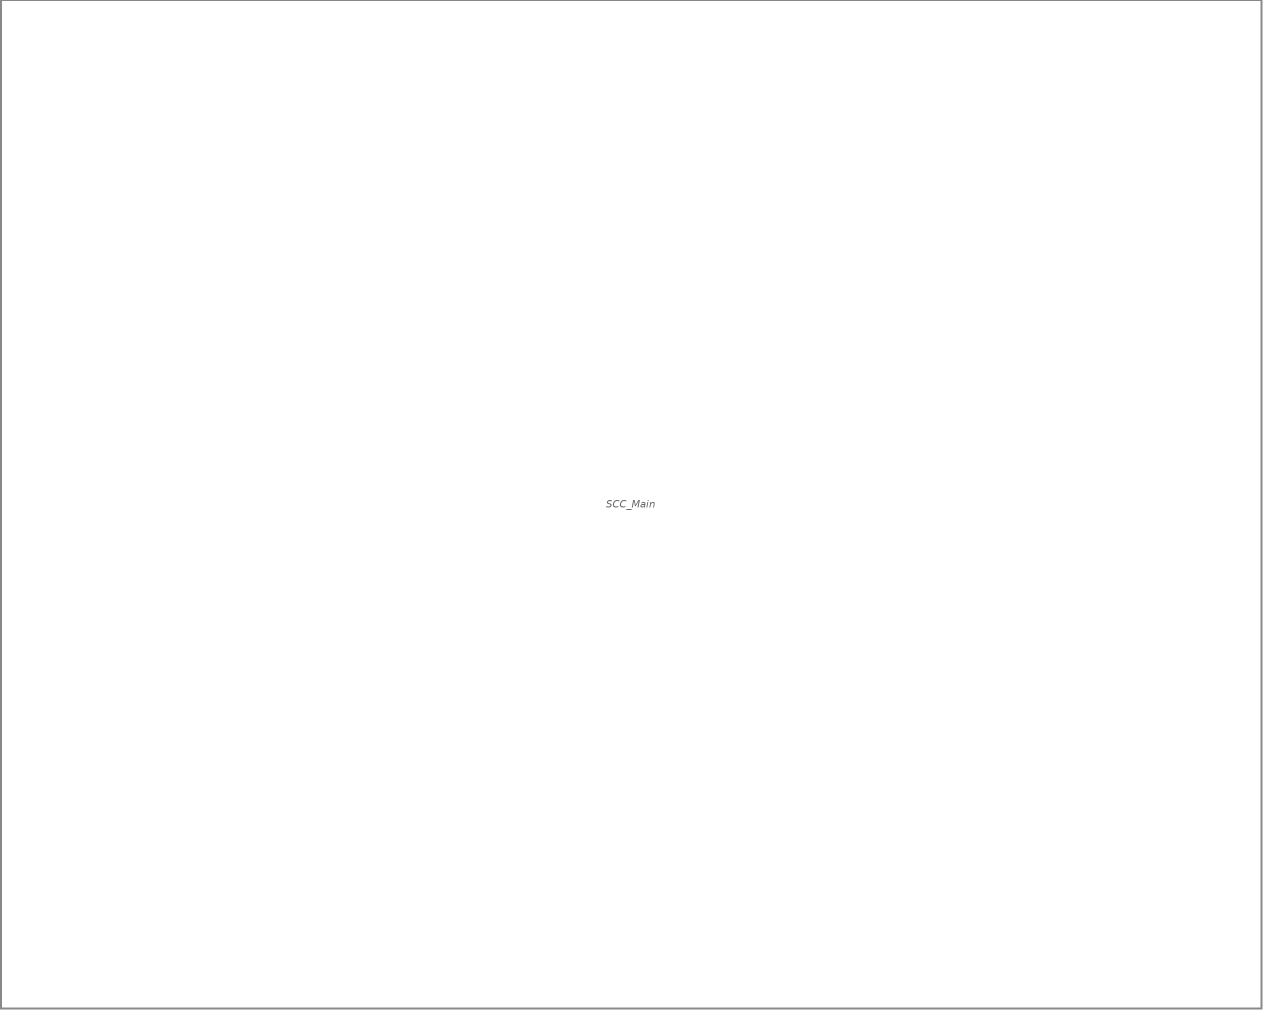
VISUALIZATION SCC  // 1263x1010
    TabControl (1,0 1260x1008)
        shows SCC_Main()
        shows SCC_activeDamping()
        [0]: TabTitle=Main
        [1]: TabTitle=Active Damping
END_VISUALIZATION
